LIN {X 0,Y 276.672,Z 702.695,A -85,B 0,C 180,E1 10836.654,E2 10836.654} C_VEL
LIN {X 0,Y 284.266,Z 684.369,A -85,B 0,C 180,E1 10834.788,E2 10834.788} C_VEL
LIN {X 0,Y 290.74,Z 666.187,A -85,B 0,C 180,E1 10833.316,E2 10833.316} C_VEL
LIN {X 0,Y 296.314,Z 647.189,A -85,B 0,C 180,E1 10832.121,E2 10832.121} C_VEL
LIN {X 0,Y 301.073,Z 626.782,A -85,B 0,C 180,E1 10831.146,E2 10831.146} C_VEL
LIN {X 0,Y 304.823,Z 604.834,A -85,B 0,C 180,E1 10830.396,E2 10830.396} C_VEL
LIN {X 0,Y 307.244,Z 581.509,A -85,B 0,C 180,E1 10829.851,E2 10829.851} C_VEL
LIN {X 0,Y 318.567,Z 436.926,A -85,B 0,C 180,E1 10826.925,E2 10826.925} C_VEL
LIN {X 0,Y 313.607,Z 427.1,A -85,B 0,C 180,E1 10824.286,E2 10824.286} C_VEL
LIN {X 0,Y 310.865,Z 421.791,A -85,B 0,C 180,E1 10822.654,E2 10822.654} C_VEL
LIN {X 0,Y 308.904,Z 419.239,A -85,B 0,C 180,E1 10821.467,E2 10821.467} C_VEL
LIN {X 0,Y 305.636,Z 417.774,A -85,B 0,C 180,E1 10819.49,E2 10819.49} C_VEL
LIN {X 0,Y 302.26,Z 416.33,A -85,B 0,C 180,E1 10817.137,E2 10817.137} C_VEL
LIN {X 0,Y 301.335,Z 415.075,A -85,B 0,C 180,E1 10816.335,E2 10816.335} C_VEL
LIN {X 0,Y 298.276,Z 409.863,A -85,B 0,C 180,E1 10813.078,E2 10813.078} C_VEL
LIN {X 0,Y 296.354,Z 406.465,A -85,B 0,C 180,E1 10810.301,E2 10810.301} C_VEL
LIN {X 0,Y 294.296,Z 402.303,A -85,B 0,C 180,E1 10804.677,E2 10804.677} C_VEL
LIN {X 0,Y 294.445,Z 402.242,A -85,B 0,C 180,E1 10799.611,E2 10799.611} C_VEL
LIN {X 0,Y 294.991,Z 403.216,A -85,B 0,C 180,E1 10797.669,E2 10797.669} C_VEL
LIN {X 0,Y 297.892,Z 407.607,A -85,B 0,C 180,E1 10792.479,E2 10792.479} C_VEL
LIN {X 0,Y 300.923,Z 412.517,A -85,B 0,C 180,E1 10789.083,E2 10789.083} C_VEL
LIN {X 0,Y 304.112,Z 417.715,A -85,B 0,C 180,E1 10786.307,E2 10786.307} C_VEL
LIN {X 0,Y 308.123,Z 424.469,A -85,B 0,C 180,E1 10783.408,E2 10783.408} C_VEL
LIN {X 0,Y 313.319,Z 434.005,A -85,B 0,C 180,E1 10780.229,E2 10780.229} C_VEL
LIN {X 0,Y 316.208,Z 439.917,A -85,B 0,C 180,E1 10778.643,E2 10778.643} C_VEL
LIN {X 0,Y 301.942,Z 602.181,A -85,B 0,C 180,E1 10775.206,E2 10775.206} C_VEL
LIN {X 0,Y 298.426,Z 624.101,A -85,B 0,C 180,E1 10774.558,E2 10774.558} C_VEL
LIN {X 0,Y 293.62,Z 645.542,A -85,B 0,C 180,E1 10773.691,E2 10773.691} C_VEL
LIN {X 0,Y 287.814,Z 666.096,A -85,B 0,C 180,E1 10772.57,E2 10772.57} C_VEL
LIN {X 0,Y 280.882,Z 686.418,A -85,B 0,C 180,E1 10771.123,E2 10771.123} C_VEL
LIN {X 0,Y 273.081,Z 705.676,A -85,B 0,C 180,E1 10769.362,E2 10769.362} C_VEL
LIN {X 0,Y 264.582,Z 724.162,A -85,B 0,C 180,E1 10767.225,E2 10767.225} C_VEL
LIN {X 0,Y 255.528,Z 741.796,A -85,B 0,C 180,E1 10764.668,E2 10764.668} C_VEL
LIN {X 0,Y 246.449,Z 757.992,A -85,B 0,C 180,E1 10761.722,E2 10761.722} C_VEL
LIN {X 0,Y 237.249,Z 773.128,A -85,B 0,C 180,E1 10758.239,E2 10758.239} C_VEL
LIN {X 0,Y 228.73,Z 786.502,A -85,B 0,C 180,E1 10754.378,E2 10754.378} C_VEL
LIN {X 0,Y 220.859,Z 798.628,A -85,B 0,C 180,E1 10750.003,E2 10750.003} C_VEL
LIN {X 0,Y 213.914,Z 809.4,A -85,B 0,C 180,E1 10745.093,E2 10745.093} C_VEL
LIN {X 0,Y 208.157,Z 818.76,A -85,B 0,C 180,E1 10739.61,E2 10739.61} C_VEL
LIN {X 0,Y 203.936,Z 826.542,A -85,B 0,C 180,E1 10733.704,E2 10733.704} C_VEL
LIN {X 0,Y 201.477,Z 832.324,A -85,B 0,C 180,E1 10727.919,E2 10727.919} C_VEL
LIN {X 0,Y 200.346,Z 836.379,A -85,B 0,C 180,E1 10722.099,E2 10722.099} C_VEL
LIN {X 0,Y 200.15,Z 838.918,A -85,B 0,C 180,E1 10716.309,E2 10716.309} C_VEL
LIN {X 0,Y 200.239,Z 839.79,A -85,B 0,C 180,E1 10711.717,E2 10711.717} C_VEL
LIN {X 0,Y 200.223,Z 839.71,A -85,B 0,C 180,E1 10707.424,E2 10707.424} C_VEL
LIN {X 0,Y 200.147,Z 838.438,A -85,B 0,C 180,E1 10702.248,E2 10702.248} C_VEL
LIN {X 0,Y 200.445,Z 835.835,A -85,B 0,C 180,E1 10697.029,E2 10697.029} C_VEL
LIN {X 0,Y 201.851,Z 831.232,A -85,B 0,C 180,E1 10690.918,E2 10690.918} C_VEL
LIN {X 0,Y 204.615,Z 825.211,A -85,B 0,C 180,E1 10685.151,E2 10685.151} C_VEL
LIN {X 0,Y 209.018,Z 817.23,A -85,B 0,C 180,E1 10679.433,E2 10679.433} C_VEL
LIN {X 0,Y 215.251,Z 807.171,A -85,B 0,C 180,E1 10673.849,E2 10673.849} C_VEL
LIN {X 0,Y 222.494,Z 796.02,A -85,B 0,C 180,E1 10668.998,E2 10668.998} C_VEL
LIN {X 0,Y 230.974,Z 782.987,A -85,B 0,C 180,E1 10664.529,E2 10664.529} C_VEL
LIN {X 0,Y 239.928,Z 768.64,A -85,B 0,C 180,E1 10660.674,E2 10660.674} C_VEL
LIN {X 0,Y 249.093,Z 753.165,A -85,B 0,C 180,E1 10657.369,E2 10657.369} C_VEL
LIN {X 0,Y 258.358,Z 736.244,A -85,B 0,C 180,E1 10654.483,E2 10654.483} C_VEL
LIN {X 0,Y 267.078,Z 718.805,A -85,B 0,C 180,E1 10652.113,E2 10652.113} C_VEL
LIN {X 0,Y 275.548,Z 699.551,A -85,B 0,C 180,E1 10650.049,E2 10650.049} C_VEL
LIN {X 0,Y 283.028,Z 679.99,A -85,B 0,C 180,E1 10648.403,E2 10648.403} C_VEL
LIN {X 0,Y 289.656,Z 659.53,A -85,B 0,C 180,E1 10647.056,E2 10647.056} C_VEL
LIN {X 0,Y 295.215,Z 638.606,A -85,B 0,C 180,E1 10646.008,E2 10646.008} C_VEL
LIN {X 0,Y 299.653,Z 616.702,A -85,B 0,C 180,E1 10645.216,E2 10645.216} C_VEL
LIN {X 0,Y 302.559,Z 594.85,A -85,B 0,C 180,E1 10644.635,E2 10644.635} C_VEL
LIN {X 0,Y 316.03,Z 439.44,A -85,B 0,C 180,E1 10641.336,E2 10641.336} C_VEL
LIN {X 0,Y 310.546,Z 428.999,A -85,B 0,C 180,E1 10638.247,E2 10638.247} C_VEL
LIN {X 0,Y 305.934,Z 420.872,A -85,B 0,C 180,E1 10635.205,E2 10635.205} C_VEL
LIN {X 0,Y 302.263,Z 414.828,A -85,B 0,C 180,E1 10632.319,E2 10632.319} C_VEL
LIN {X 0,Y 299.8,Z 410.85,A -85,B 0,C 180,E1 10629.987,E2 10629.987} C_VEL
LIN {X 0,Y 297.263,Z 406.753,A -85,B 0,C 180,E1 10626.955,E2 10626.955} C_VEL
LIN {X 0,Y 294.455,Z 402.282,A -85,B 0,C 180,E1 10621.362,E2 10621.362} C_VEL
LIN {X 0,Y 293.88,Z 401.961,A -85,B 0,C 180,E1 10616.489,E2 10616.489} C_VEL
LIN {X 0,Y 294.254,Z 402.624,A -85,B 0,C 180,E1 10614.149,E2 10614.149} C_VEL
LIN {X 0,Y 296.669,Z 407.215,A -85,B 0,C 180,E1 10608.727,E2 10608.727} C_VEL
LIN {X 0,Y 299.047,Z 411.383,A -85,B 0,C 180,E1 10605.675,E2 10605.675} C_VEL
LIN {X 0,Y 301.903,Z 416.413,A -85,B 0,C 180,E1 10602.857,E2 10602.857} C_VEL
LIN {X 0,Y 305.778,Z 423.433,A -85,B 0,C 180,E1 10599.774,E2 10599.774} C_VEL
LIN {X 0,Y 310.068,Z 431.486,A -85,B 0,C 180,E1 10596.933,E2 10596.933} C_VEL
LIN {X 0,Y 314.826,Z 441.211,A -85,B 0,C 180,E1 10594.2,E2 10594.2} C_VEL
LIN {X 0,Y 301.88,Z 598.214,A -85,B 0,C 180,E1 10591.019,E2 10591.019} C_VEL
LIN {X 0,Y 298.541,Z 619.734,A -85,B 0,C 180,E1 10590.375,E2 10590.375} C_VEL
LIN {X 0,Y 294.115,Z 639.956,A -85,B 0,C 180,E1 10589.515,E2 10589.515} C_VEL
LIN {X 0,Y 288.351,Z 660.439,A -85,B 0,C 180,E1 10588.348,E2 10588.348} C_VEL
LIN {X 0,Y 282.015,Z 678.968,A -85,B 0,C 180,E1 10586.978,E2 10586.978} C_VEL
LIN {X 0,Y 274.458,Z 697.523,A -85,B 0,C 180,E1 10585.231,E2 10585.231} C_VEL
LIN {X 0,Y 266.516,Z 714.386,A -85,B 0,C 180,E1 10583.22,E2 10583.22} C_VEL
LIN {X 0,Y 257.664,Z 731.079,A -85,B 0,C 180,E1 10580.727,E2 10580.727} C_VEL
LIN {X 0,Y 249.019,Z 745.804,A -85,B 0,C 180,E1 10577.97,E2 10577.97} C_VEL
LIN {X 0,Y 240.155,Z 759.6,A -85,B 0,C 180,E1 10574.716,E2 10574.716} C_VEL
LIN {X 0,Y 231.593,Z 771.968,A -85,B 0,C 180,E1 10571.012,E2 10571.012} C_VEL
LIN {X 0,Y 223.172,Z 783.563,A -85,B 0,C 180,E1 10566.573,E2 10566.573} C_VEL
LIN {X 0,Y 216.051,Z 793.13,A -85,B 0,C 180,E1 10561.841,E2 10561.841} C_VEL
LIN {X 0,Y 210.056,Z 801.285,A -85,B 0,C 180,E1 10556.578,E2 10556.578} C_VEL
LIN {X 0,Y 205.429,Z 807.855,A -85,B 0,C 180,E1 10550.811,E2 10550.811} C_VEL
LIN {X 0,Y 202.547,Z 812.407,A -85,B 0,C 180,E1 10545.166,E2 10545.166} C_VEL
LIN {X 0,Y 200.948,Z 815.59,A -85,B 0,C 180,E1 10539.162,E2 10539.162} C_VEL
LIN {X 0,Y 200.4,Z 817.13,A -85,B 0,C 180,E1 10533.719,E2 10533.719} C_VEL
LIN {X 0,Y 200.332,Z 817.331,A -85,B 0,C 180,E1 10528.284,E2 10528.284} C_VEL
LIN {X 0,Y 200.659,Z 816.383,A -85,B 0,C 180,E1 10522.844,E2 10522.844} C_VEL
LIN {X 0,Y 201.767,Z 813.901,A -85,B 0,C 180,E1 10517.115,E2 10517.115} C_VEL
LIN {X 0,Y 204.211,Z 809.715,A -85,B 0,C 180,E1 10511.147,E2 10511.147} C_VEL
LIN {X 0,Y 208.255,Z 803.795,A -85,B 0,C 180,E1 10505.311,E2 10505.311} C_VEL
LIN {X 0,Y 213.728,Z 796.374,A -85,B 0,C 180,E1 10499.937,E2 10499.937} C_VEL
LIN {X 0,Y 220.68,Z 787.067,A -85,B 0,C 180,E1 10494.873,E2 10494.873} C_VEL
LIN {X 0,Y 228.684,Z 776.16,A -85,B 0,C 180,E1 10490.333,E2 10490.333} C_VEL
LIN {X 0,Y 237.414,Z 763.748,A -85,B 0,C 180,E1 10486.318,E2 10486.318} C_VEL
LIN {X 0,Y 246.597,Z 749.809,A -85,B 0,C 180,E1 10482.789,E2 10482.789} C_VEL
LIN {X 0,Y 255.391,Z 735.349,A -85,B 0,C 180,E1 10479.886,E2 10479.886} C_VEL
LIN {X 0,Y 264.448,Z 718.812,A -85,B 0,C 180,E1 10477.263,E2 10477.263} C_VEL
LIN {X 0,Y 272.637,Z 701.841,A -85,B 0,C 180,E1 10475.135,E2 10475.135} C_VEL
LIN {X 0,Y 280.359,Z 683.561,A -85,B 0,C 180,E1 10473.314,E2 10473.314} C_VEL
LIN {X 0,Y 287.141,Z 664.723,A -85,B 0,C 180,E1 10471.831,E2 10471.831} C_VEL
LIN {X 0,Y 293.069,Z 644.824,A -85,B 0,C 180,E1 10470.619,E2 10470.619} C_VEL
LIN {X 0,Y 297.928,Z 623.713,A -85,B 0,C 180,E1 10469.666,E2 10469.666} C_VEL
LIN {X 0,Y 301.373,Z 603.001,A -85,B 0,C 180,E1 10469.003,E2 10469.003} C_VEL
LIN {X 0,Y 304.114,Z 575.028,A -85,B 0,C 180,E1 10468.38,E2 10468.38} C_VEL
LIN {X 0,Y 314.952,Z 441.247,A -85,B 0,C 180,E1 10465.68,E2 10465.68} C_VEL
LIN {X 0,Y 309.851,Z 430.902,A -85,B 0,C 180,E1 10462.732,E2 10462.732} C_VEL
LIN {X 0,Y 305.331,Z 422.359,A -85,B 0,C 180,E1 10459.663,E2 10459.663} C_VEL
LIN {X 0,Y 301.335,Z 415.075,A -85,B 0,C 180,E1 10456.335,E2 10456.335} C_VEL
LIN {X 0,Y 299.91,Z 413.527,A -85,B 0,C 180,E1 10455.028,E2 10455.028} C_VEL
LIN {X 0,Y 297.669,Z 413.637,A -85,B 0,C 180,E1 10452.932,E2 10452.932} C_VEL
LIN {X 0,Y 295.352,Z 414.27,A -85,B 0,C 180,E1 10450.238,E2 10450.238} C_VEL
LIN {X 0,Y 294.955,Z 413.941,A -85,B 0,C 180,E1 10449.588,E2 10449.588} C_VEL
LIN {X 0,Y 293.289,Z 410.213,A -85,B 0,C 180,E1 10444.498,E2 10444.498} C_VEL
LIN {X 0,Y 293.469,Z 410.189,A -85,B 0,C 180,E1 10439.61,E2 10439.61} C_VEL
LIN {X 0,Y 293.995,Z 411.255,A -85,B 0,C 180,E1 10437.661,E2 10437.661} C_VEL
LIN {X 0,Y 296.603,Z 415.287,A -85,B 0,C 180,E1 10432.835,E2 10432.835} C_VEL
LIN {X 0,Y 299.526,Z 420.223,A -85,B 0,C 180,E1 10429.421,E2 10429.421} C_VEL
LIN {X 0,Y 302.511,Z 425.254,A -85,B 0,C 180,E1 10426.72,E2 10426.72} C_VEL
LIN {X 0,Y 306.399,Z 432.083,A -85,B 0,C 180,E1 10423.799,E2 10423.799} C_VEL
LIN {X 0,Y 311.167,Z 441.169,A -85,B 0,C 180,E1 10420.771,E2 10420.771} C_VEL
LIN {X 0,Y 312.661,Z 444.381,A -85,B 0,C 180,E1 10419.895,E2 10419.895} C_VEL
LIN {X 0,Y 298.397,Z 602.136,A -85,B 0,C 180,E1 10416.579,E2 10416.579} C_VEL
LIN {X 0,Y 294.778,Z 624.153,A -85,B 0,C 180,E1 10415.937,E2 10415.937} C_VEL
LIN {X 0,Y 289.915,Z 645.311,A -85,B 0,C 180,E1 10415.095,E2 10415.095} C_VEL
LIN {X 0,Y 284.02,Z 665.699,A -85,B 0,C 180,E1 10414.003,E2 10414.003} C_VEL
LIN {X 0,Y 277.026,Z 685.694,A -85,B 0,C 180,E1 10412.605,E2 10412.605} C_VEL
LIN {X 0,Y 268.993,Z 705.031,A -85,B 0,C 180,E1 10410.866,E2 10410.866} C_VEL
LIN {X 0,Y 260.257,Z 723.497,A -85,B 0,C 180,E1 10408.759,E2 10408.759} C_VEL
LIN {X 0,Y 251.17,Z 740.681,A -85,B 0,C 180,E1 10406.301,E2 10406.301} C_VEL
LIN {X 0,Y 241.439,Z 757.416,A -85,B 0,C 180,E1 10403.275,E2 10403.275} C_VEL
LIN {X 0,Y 231.794,Z 772.617,A -85,B 0,C 180,E1 10399.772,E2 10399.772} C_VEL
LIN {X 0,Y 222.858,Z 786.007,A -85,B 0,C 180,E1 10395.875,E2 10395.875} C_VEL
LIN {X 0,Y 214.358,Z 798.4,A -85,B 0,C 180,E1 10391.326,E2 10391.326} C_VEL
LIN {X 0,Y 206.806,Z 809.455,A -85,B 0,C 180,E1 10386.145,E2 10386.145} C_VEL
LIN {X 0,Y 200.684,Z 818.756,A -85,B 0,C 180,E1 10380.467,E2 10380.467} C_VEL
LIN {X 0,Y 196.215,Z 826.398,A -85,B 0,C 180,E1 10374.377,E2 10374.377} C_VEL
LIN {X 0,Y 193.482,Z 832.327,A -85,B 0,C 180,E1 10368.039,E2 10368.039} C_VEL
LIN {X 0,Y 192.362,Z 836.119,A -85,B 0,C 180,E1 10362.265,E2 10362.265} C_VEL
LIN {X 0,Y 192.16,Z 838.516,A -85,B 0,C 180,E1 10356.377,E2 10356.377} C_VEL
LIN {X 0,Y 192.25,Z 839.342,A -85,B 0,C 180,E1 10351.788,E2 10351.788} C_VEL
LIN {X 0,Y 192.232,Z 839.261,A -85,B 0,C 180,E1 10347.317,E2 10347.317} C_VEL
LIN {X 0,Y 192.155,Z 837.984,A -85,B 0,C 180,E1 10341.924,E2 10341.924} C_VEL
LIN {X 0,Y 192.511,Z 835.376,A -85,B 0,C 180,E1 10336.484,E2 10336.484} C_VEL
LIN {X 0,Y 194.094,Z 830.766,A -85,B 0,C 180,E1 10330.124,E2 10330.124} C_VEL
LIN {X 0,Y 197.134,Z 824.742,A -85,B 0,C 180,E1 10324.14,E2 10324.14} C_VEL
LIN {X 0,Y 201.816,Z 816.888,A -85,B 0,C 180,E1 10318.322,E2 10318.322} C_VEL
LIN {X 0,Y 208.214,Z 807.226,A -85,B 0,C 180,E1 10312.768,E2 10312.768} C_VEL
LIN {X 0,Y 215.835,Z 796.186,A -85,B 0,C 180,E1 10307.802,E2 10307.802} C_VEL
LIN {X 0,Y 224.689,Z 783.24,A -85,B 0,C 180,E1 10303.258,E2 10303.258} C_VEL
LIN {X 0,Y 234.032,Z 768.997,A -85,B 0,C 180,E1 10299.352,E2 10299.352} C_VEL
LIN {X 0,Y 243.538,Z 753.667,A -85,B 0,C 180,E1 10296.024,E2 10296.024} C_VEL
LIN {X 0,Y 252.791,Z 737.538,A -85,B 0,C 180,E1 10293.226,E2 10293.226} C_VEL
LIN {X 0,Y 261.927,Z 719.945,A -85,B 0,C 180,E1 10290.81,E2 10290.81} C_VEL
LIN {X 0,Y 270.412,Z 701.461,A -85,B 0,C 180,E1 10288.802,E2 10288.802} C_VEL
LIN {X 0,Y 278.49,Z 681.282,A -85,B 0,C 180,E1 10287.081,E2 10287.081} C_VEL
LIN {X 0,Y 285.281,Z 661.235,A -85,B 0,C 180,E1 10285.748,E2 10285.748} C_VEL
LIN {X 0,Y 291.071,Z 640.344,A -85,B 0,C 180,E1 10284.693,E2 10284.693} C_VEL
LIN {X 0,Y 295.632,Z 618.832,A -85,B 0,C 180,E1 10283.908,E2 10283.908} C_VEL
LIN {X 0,Y 298.847,Z 596.481,A -85,B 0,C 180,E1 10283.303,E2 10283.303} C_VEL
LIN {X 0,Y 312.496,Z 443.973,A -85,B 0,C 180,E1 10280.093,E2 10280.093} C_VEL
LIN {X 0,Y 307.033,Z 433.38,A -85,B 0,C 180,E1 10276.75,E2 10276.75} C_VEL
LIN {X 0,Y 302.666,Z 425.671,A -85,B 0,C 180,E1 10273.565,E2 10273.565} C_VEL
LIN {X 0,Y 300.202,Z 421.559,A -85,B 0,C 180,E1 10271.43,E2 10271.43} C_VEL
LIN {X 0,Y 298.341,Z 418.411,A -85,B 0,C 180,E1 10269.549,E2 10269.549} C_VEL
LIN {X 0,Y 295.99,Z 414.475,A -85,B 0,C 180,E1 10266.595,E2 10266.595} C_VEL
LIN {X 0,Y 293.418,Z 410.184,A -85,B 0,C 180,E1 10261.171,E2 10261.171} C_VEL
LIN {X 0,Y 292.92,Z 409.93,A -85,B 0,C 180,E1 10256.281,E2 10256.281} C_VEL
LIN {X 0,Y 293.277,Z 410.644,A -85,B 0,C 180,E1 10254.129,E2 10254.129} C_VEL
LIN {X 0,Y 295.499,Z 415.05,A -85,B 0,C 180,E1 10248.978,E2 10248.978} C_VEL
LIN {X 0,Y 297.683,Z 419.005,A -85,B 0,C 180,E1 10246.067,E2 10246.067} C_VEL
LIN {X 0,Y 300.402,Z 423.986,A -85,B 0,C 180,E1 10243.267,E2 10243.267} C_VEL
LIN {X 0,Y 304.105,Z 430.961,A -85,B 0,C 180,E1 10240.205,E2 10240.205} C_VEL
LIN {X 0,Y 308.117,Z 438.851,A -85,B 0,C 180,E1 10237.435,E2 10237.435} C_VEL
LIN {X 0,Y 311.346,Z 445.782,A -85,B 0,C 180,E1 10235.461,E2 10235.461} C_VEL
LIN {X 0,Y 298.336,Z 598.392,A -85,B 0,C 180,E1 10232.39,E2 10232.39} C_VEL
LIN {X 0,Y 294.913,Z 619.881,A -85,B 0,C 180,E1 10231.754,E2 10231.754} C_VEL
LIN {X 0,Y 290.352,Z 640.196,A -85,B 0,C 180,E1 10230.902,E2 10230.902} C_VEL
LIN {X 0,Y 284.254,Z 661.228,A -85,B 0,C 180,E1 10229.714,E2 10229.714} C_VEL
LIN {X 0,Y 277.387,Z 680.531,A -85,B 0,C 180,E1 10228.283,E2 10228.283} C_VEL
LIN {X 0,Y 269.638,Z 698.933,A -85,B 0,C 180,E1 10226.544,E2 10226.544} C_VEL
LIN {X 0,Y 261.13,Z 716.273,A -85,B 0,C 180,E1 10224.452,E2 10224.452} C_VEL
LIN {X 0,Y 252.017,Z 732.702,A -85,B 0,C 180,E1 10221.953,E2 10221.953} C_VEL
LIN {X 0,Y 242.501,Z 748.118,A -85,B 0,C 180,E1 10218.982,E2 10218.982} C_VEL
LIN {X 0,Y 233.387,Z 761.659,A -85,B 0,C 180,E1 10215.678,E2 10215.678} C_VEL
LIN {X 0,Y 224.074,Z 774.491,A -85,B 0,C 180,E1 10211.67,E2 10211.67} C_VEL
LIN {X 0,Y 215.443,Z 785.693,A -85,B 0,C 180,E1 10207.107,E2 10207.107} C_VEL
LIN {X 0,Y 208.146,Z 794.915,A -85,B 0,C 180,E1 10202.221,E2 10202.221} C_VEL
LIN {X 0,Y 201.748,Z 803.09,A -85,B 0,C 180,E1 10196.489,E2 10196.489} C_VEL
LIN {X 0,Y 197.317,Z 809.099,A -85,B 0,C 180,E1 10190.775,E2 10190.775} C_VEL
LIN {X 0,Y 194.333,Z 813.638,A -85,B 0,C 180,E1 10184.602,E2 10184.602} C_VEL
LIN {X 0,Y 192.875,Z 816.357,A -85,B 0,C 180,E1 10178.646,E2 10178.646} C_VEL
LIN {X 0,Y 192.376,Z 817.707,A -85,B 0,C 180,E1 10172.681,E2 10172.681} C_VEL
LIN {X 0,Y 192.36,Z 817.738,A -85,B 0,C 180,E1 10167.617,E2 10167.617} C_VEL
LIN {X 0,Y 192.82,Z 816.515,A -85,B 0,C 180,E1 10161.652,E2 10161.652} C_VEL
LIN {X 0,Y 194.206,Z 813.905,A -85,B 0,C 180,E1 10155.693,E2 10155.693} C_VEL
LIN {X 0,Y 197.084,Z 809.449,A -85,B 0,C 180,E1 10149.51,E2 10149.51} C_VEL
LIN {X 0,Y 201.68,Z 803.242,A -85,B 0,C 180,E1 10143.501,E2 10143.501} C_VEL
LIN {X 0,Y 208.081,Z 795.087,A -85,B 0,C 180,E1 10137.749,E2 10137.749} C_VEL
LIN {X 0,Y 215.341,Z 785.936,A -85,B 0,C 180,E1 10132.872,E2 10132.872} C_VEL
LIN {X 0,Y 223.961,Z 774.775,A -85,B 0,C 180,E1 10128.304,E2 10128.304} C_VEL
LIN {X 0,Y 233.265,Z 761.979,A -85,B 0,C 180,E1 10124.291,E2 10124.291} C_VEL
LIN {X 0,Y 242.368,Z 748.5,A -85,B 0,C 180,E1 10120.982,E2 10120.982} C_VEL
LIN {X 0,Y 252.198,Z 732.614,A -85,B 0,C 180,E1 10117.915,E2 10117.915} C_VEL
LIN {X 0,Y 260.995,Z 716.818,A -85,B 0,C 180,E1 10115.506,E2 10115.506} C_VEL
LIN {X 0,Y 269.497,Z 699.536,A -85,B 0,C 180,E1 10113.411,E2 10113.411} C_VEL
LIN {X 0,Y 277.246,Z 681.252,A -85,B 0,C 180,E1 10111.67,E2 10111.67} C_VEL
LIN {X 0,Y 284.112,Z 662.135,A -85,B 0,C 180,E1 10110.237,E2 10110.237} C_VEL
LIN {X 0,Y 290.004,Z 642.19,A -85,B 0,C 180,E1 10109.087,E2 10109.087} C_VEL
LIN {X 0,Y 294.803,Z 621.393,A -85,B 0,C 180,E1 10108.192,E2 10108.192} C_VEL
LIN {X 0,Y 298.306,Z 599.8,A -85,B 0,C 180,E1 10107.541,E2 10107.541} C_VEL
LIN {X 0,Y 302.156,Z 556.981,A -85,B 0,C 180,E1 10106.647,E2 10106.647} C_VEL
LIN {X 0,Y 311.488,Z 445.629,A -85,B 0,C 180,E1 10104.411,E2 10104.411} C_VEL
LIN {X 0,Y 306.307,Z 434.97,A -85,B 0,C 180,E1 10101.143,E2 10101.143} C_VEL
LIN {X 0,Y 302.014,Z 426.745,A -85,B 0,C 180,E1 10097.883,E2 10097.883} C_VEL
LIN {X 0,Y 299.225,Z 421.673,A -85,B 0,C 180,E1 10095.307,E2 10095.307} C_VEL
LIN {X 0,Y 296.924,Z 417.455,A -85,B 0,C 180,E1 10092.644,E2 10092.644} C_VEL
LIN {X 0,Y 295.16,Z 414.211,A -85,B 0,C 180,E1 10089.949,E2 10089.949} C_VEL
LIN {X 0,Y 294.955,Z 413.941,A -85,B 0,C 180,E1 10089.588,E2 10089.588} C_VEL
LIN {X 0,Y 294.052,Z 413.81,A -85,B 0,C 180,E1 10087.976,E2 10087.976} C_VEL
LIN {X 0,Y 292.202,Z 417.825,A -85,B 0,C 180,E1 10083.327,E2 10083.327} C_VEL
LIN {X 0,Y 292.155,Z 417.945,A -85,B 0,C 180,E1 10082.665,E2 10082.665} C_VEL
LIN {X 0,Y 292.731,Z 418.491,A -85,B 0,C 180,E1 10078.63,E2 10078.63} C_VEL
LIN {X 0,Y 295.393,Z 423.114,A -85,B 0,C 180,E1 10073.099,E2 10073.099} C_VEL
LIN {X 0,Y 298.141,Z 427.926,A -85,B 0,C 180,E1 10069.762,E2 10069.762} C_VEL
LIN {X 0,Y 301.142,Z 433.176,A -85,B 0,C 180,E1 10066.952,E2 10066.952} C_VEL
LIN {X 0,Y 305.407,Z 441.02,A -85,B 0,C 180,E1 10063.696,E2 10063.696} C_VEL
LIN {X 0,Y 309.261,Z 448.958,A -85,B 0,C 180,E1 10061.174,E2 10061.174} C_VEL
LIN {X 0,Y 295.041,Z 601.989,A -85,B 0,C 180,E1 10057.987,E2 10057.987} C_VEL
LIN {X 0,Y 291.349,Z 623.97,A -85,B 0,C 180,E1 10057.357,E2 10057.357} C_VEL
LIN {X 0,Y 286.539,Z 644.522,A -85,B 0,C 180,E1 10056.56,E2 10056.56} C_VEL
LIN {X 0,Y 280.683,Z 664.509,A -85,B 0,C 180,E1 10055.523,E2 10055.523} C_VEL
LIN {X 0,Y 273.361,Z 684.962,A -85,B 0,C 180,E1 10054.126,E2 10054.126} C_VEL
LIN {X 0,Y 265.466,Z 703.562,A -85,B 0,C 180,E1 10052.495,E2 10052.495} C_VEL
LIN {X 0,Y 256.046,Z 722.99,A -85,B 0,C 180,E1 10050.324,E2 10050.324} C_VEL
LIN {X 0,Y 246.684,Z 740.136,A -85,B 0,C 180,E1 10047.897,E2 10047.897} C_VEL
LIN {X 0,Y 236.816,Z 756.502,A -85,B 0,C 180,E1 10044.957,E2 10044.957} C_VEL
LIN {X 0,Y 227.099,Z 771.235,A -85,B 0,C 180,E1 10041.597,E2 10041.597} C_VEL
LIN {X 0,Y 217.143,Z 785.515,A -85,B 0,C 180,E1 10037.452,E2 10037.452} C_VEL
LIN {X 0,Y 208.368,Z 797.663,A -85,B 0,C 180,E1 10032.951,E2 10032.951} C_VEL
LIN {X 0,Y 200.139,Z 808.976,A -85,B 0,C 180,E1 10027.551,E2 10027.551} C_VEL
LIN {X 0,Y 193.629,Z 818.185,A -85,B 0,C 180,E1 10021.782,E2 10021.782} C_VEL
LIN {X 0,Y 188.712,Z 825.932,A -85,B 0,C 180,E1 10015.414,E2 10015.414} C_VEL
LIN {X 0,Y 185.697,Z 831.849,A -85,B 0,C 180,E1 10008.848,E2 10008.848} C_VEL
LIN {X 0,Y 184.423,Z 835.639,A -85,B 0,C 180,E1 10002.843,E2 10002.843} C_VEL
LIN {X 0,Y 184.172,Z 838.016,A -85,B 0,C 180,E1 9996.859,E2 9996.859} C_VEL
LIN {X 0,Y 184.26,Z 838.893,A -85,B 0,C 180,E1 9991.866,E2 9991.866} C_VEL
LIN {X 0,Y 184.241,Z 838.812,A -85,B 0,C 180,E1 9987.201,E2 9987.201} C_VEL
LIN {X 0,Y 184.164,Z 837.53,A -85,B 0,C 180,E1 9981.571,E2 9981.571} C_VEL
LIN {X 0,Y 184.6,Z 834.875,A -85,B 0,C 180,E1 9975.816,E2 9975.816} C_VEL
LIN {X 0,Y 186.377,Z 830.302,A -85,B 0,C 180,E1 9969.264,E2 9969.264} C_VEL
LIN {X 0,Y 189.922,Z 823.931,A -85,B 0,C 180,E1 9962.742,E2 9962.742} C_VEL
LIN {X 0,Y 195.389,Z 815.559,A -85,B 0,C 180,E1 9956.451,E2 9956.451} C_VEL
LIN {X 0,Y 202.418,Z 805.667,A -85,B 0,C 180,E1 9950.784,E2 9950.784} C_VEL
LIN {X 0,Y 211.142,Z 793.712,A -85,B 0,C 180,E1 9945.506,E2 9945.506} C_VEL
LIN {X 0,Y 220.329,Z 780.934,A -85,B 0,C 180,E1 9941.124,E2 9941.124} C_VEL
LIN {X 0,Y 230.061,Z 766.742,A -85,B 0,C 180,E1 9937.316,E2 9937.316} C_VEL
LIN {X 0,Y 239.727,Z 751.568,A -85,B 0,C 180,E1 9934.118,E2 9934.118} C_VEL
LIN {X 0,Y 249.731,Z 734.476,A -85,B 0,C 180,E1 9931.265,E2 9931.265} C_VEL
LIN {X 0,Y 258.926,Z 717.112,A -85,B 0,C 180,E1 9928.976,E2 9928.976} C_VEL
LIN {X 0,Y 267.687,Z 698.335,A -85,B 0,C 180,E1 9927.024,E2 9927.024} C_VEL
LIN {X 0,Y 275.285,Z 679.439,A -85,B 0,C 180,E1 9925.486,E2 9925.486} C_VEL
LIN {X 0,Y 282.234,Z 659.05,A -85,B 0,C 180,E1 9924.187,E2 9924.187} C_VEL
LIN {X 0,Y 288.035,Z 638.224,A -85,B 0,C 180,E1 9923.183,E2 9923.183} C_VEL
LIN {X 0,Y 292.661,Z 616.369,A -85,B 0,C 180,E1 9922.421,E2 9922.421} C_VEL
LIN {X 0,Y 295.703,Z 594.476,A -85,B 0,C 180,E1 9921.854,E2 9921.854} C_VEL
LIN {X 0,Y 309.094,Z 448.662,A -85,B 0,C 180,E1 9918.824,E2 9918.824} C_VEL
LIN {X 0,Y 304.463,Z 439.409,A -85,B 0,C 180,E1 9915.768,E2 9915.768} C_VEL
LIN {X 0,Y 300.631,Z 432.429,A -85,B 0,C 180,E1 9912.777,E2 9912.777} C_VEL
LIN {X 0,Y 297.251,Z 426.439,A -85,B 0,C 180,E1 9909.486,E2 9909.486} C_VEL
LIN {X 0,Y 294.73,Z 422.195,A -85,B 0,C 180,E1 9906.232,E2 9906.232} C_VEL
LIN {X 0,Y 292.385,Z 418.086,A -85,B 0,C 180,E1 9900.979,E2 9900.979} C_VEL
LIN {X 0,Y 291.947,Z 417.874,A -85,B 0,C 180,E1 9896.269,E2 9896.269} C_VEL
LIN {X 0,Y 292.256,Z 418.529,A -85,B 0,C 180,E1 9894.306,E2 9894.306} C_VEL
LIN {X 0,Y 294.284,Z 422.75,A -85,B 0,C 180,E1 9889.329,E2 9889.329} C_VEL
LIN {X 0,Y 296.348,Z 426.669,A -85,B 0,C 180,E1 9886.438,E2 9886.438} C_VEL
LIN {X 0,Y 298.916,Z 431.556,A -85,B 0,C 180,E1 9883.681,E2 9883.681} C_VEL
LIN {X 0,Y 302.378,Z 438.355,A -85,B 0,C 180,E1 9880.69,E2 9880.69} C_VEL
LIN {X 0,Y 306.124,Z 446.059,A -85,B 0,C 180,E1 9877.988,E2 9877.988} C_VEL
LIN {X 0,Y 308.018,Z 450.255,A -85,B 0,C 180,E1 9876.755,E2 9876.755} C_VEL
LIN {X 0,Y 294.99,Z 598.371,A -85,B 0,C 180,E1 9873.796,E2 9873.796} C_VEL
LIN {X 0,Y 291.512,Z 619.754,A -85,B 0,C 180,E1 9873.175,E2 9873.175} C_VEL
LIN {X 0,Y 286.956,Z 639.699,A -85,B 0,C 180,E1 9872.359,E2 9872.359} C_VEL
LIN {X 0,Y 281.08,Z 659.775,A -85,B 0,C 180,E1 9871.262,E2 9871.262} C_VEL
LIN {X 0,Y 274.221,Z 678.933,A -85,B 0,C 180,E1 9869.898,E2 9869.898} C_VEL
LIN {X 0,Y 266.379,Z 697.18,A -85,B 0,C 180,E1 9868.228,E2 9868.228} C_VEL
LIN {X 0,Y 257.925,Z 714.221,A -85,B 0,C 180,E1 9866.253,E2 9866.253} C_VEL
LIN {X 0,Y 248.458,Z 731.057,A -85,B 0,C 180,E1 9863.788,E2 9863.788} C_VEL
LIN {X 0,Y 239.157,Z 745.908,A -85,B 0,C 180,E1 9861.041,E2 9861.041} C_VEL
LIN {X 0,Y 228.961,Z 760.595,A -85,B 0,C 180,E1 9857.561,E2 9857.561} C_VEL
LIN {X 0,Y 219.639,Z 772.931,A -85,B 0,C 180,E1 9853.783,E2 9853.783} C_VEL
LIN {X 0,Y 210.452,Z 784.409,A -85,B 0,C 180,E1 9849.247,E2 9849.247} C_VEL
LIN {X 0,Y 202.449,Z 794.056,A -85,B 0,C 180,E1 9844.264,E2 9844.264} C_VEL
LIN {X 0,Y 195.685,Z 802.201,A -85,B 0,C 180,E1 9838.704,E2 9838.704} C_VEL
LIN {X 0,Y 190.376,Z 808.771,A -85,B 0,C 180,E1 9832.544,E2 9832.544} C_VEL
LIN {X 0,Y 186.885,Z 813.511,A -85,B 0,C 180,E1 9826.153,E2 9826.153} C_VEL
LIN {X 0,Y 185.048,Z 816.597,A -85,B 0,C 180,E1 9819.642,E2 9819.642} C_VEL
LIN {X 0,Y 184.426,Z 818.088,A -85,B 0,C 180,E1 9813.73,E2 9813.73} C_VEL
LIN {X 0,Y 184.36,Z 818.227,A -85,B 0,C 180,E1 9808.135,E2 9808.135} C_VEL
LIN {X 0,Y 184.757,Z 817.283,A -85,B 0,C 180,E1 9802.225,E2 9802.225} C_VEL
LIN {X 0,Y 186.089,Z 814.803,A -85,B 0,C 180,E1 9796.008,E2 9796.008} C_VEL
LIN {X 0,Y 188.967,Z 810.623,A -85,B 0,C 180,E1 9789.561,E2 9789.561} C_VEL
LIN {X 0,Y 193.665,Z 804.674,A -85,B 0,C 180,E1 9783.275,E2 9783.275} C_VEL
LIN {X 0,Y 199.818,Z 797.337,A -85,B 0,C 180,E1 9777.629,E2 9777.629} C_VEL
LIN {X 0,Y 207.625,Z 787.991,A -85,B 0,C 180,E1 9772.296,E2 9772.296} C_VEL
LIN {X 0,Y 216.147,Z 777.485,A -85,B 0,C 180,E1 9767.743,E2 9767.743} C_VEL
LIN {X 0,Y 225.443,Z 765.461,A -85,B 0,C 180,E1 9763.706,E2 9763.706} C_VEL
LIN {X 0,Y 234.731,Z 752.618,A -85,B 0,C 180,E1 9760.32,E2 9760.32} C_VEL
LIN {X 0,Y 244.738,Z 737.439,A -85,B 0,C 180,E1 9757.19,E2 9757.19} C_VEL
LIN {X 0,Y 254.023,Z 721.691,A -85,B 0,C 180,E1 9754.652,E2 9754.652} C_VEL
LIN {X 0,Y 263.04,Z 704.47,A -85,B 0,C 180,E1 9752.453,E2 9752.453} C_VEL
LIN {X 0,Y 271.313,Z 686.358,A -85,B 0,C 180,E1 9750.629,E2 9750.629} C_VEL
LIN {X 0,Y 278.699,Z 667.385,A -85,B 0,C 180,E1 9749.126,E2 9749.126} C_VEL
LIN {X 0,Y 285.105,Z 647.198,A -85,B 0,C 180,E1 9747.904,E2 9747.904} C_VEL
LIN {X 0,Y 290.193,Z 626.832,A -85,B 0,C 180,E1 9746.979,E2 9746.979} C_VEL
LIN {X 0,Y 294.187,Z 605.052,A -85,B 0,C 180,E1 9746.272,E2 9746.272} C_VEL
LIN {X 0,Y 296.85,Z 581.323,A -85,B 0,C 180,E1 9745.734,E2 9745.734} C_VEL
LIN {X 0,Y 308.162,Z 450.154,A -85,B 0,C 180,E1 9743.116,E2 9743.116} C_VEL
LIN {X 0,Y 303.521,Z 440.303,A -85,B 0,C 180,E1 9739.935,E2 9739.935} C_VEL
LIN {X 0,Y 299.695,Z 432.82,A -85,B 0,C 180,E1 9736.769,E2 9736.769} C_VEL
LIN {X 0,Y 297.446,Z 428.647,A -85,B 0,C 180,E1 9734.516,E2 9734.516} C_VEL
LIN {X 0,Y 295.662,Z 425.157,A -85,B 0,C 180,E1 9732.302,E2 9732.302} C_VEL
LIN {X 0,Y 293.977,Z 421.954,A -85,B 0,C 180,E1 9729.594,E2 9729.594} C_VEL
LIN {X 0,Y 292.285,Z 418.126,A -85,B 0,C 180,E1 9724.316,E2 9724.316} C_VEL
LIN {X 0,Y 292.155,Z 417.945,A -85,B 0,C 180,E1 9722.665,E2 9722.665} C_VEL
LIN {X 0,Y 292.101,Z 418.899,A -85,B 0,C 180,E1 9721.264,E2 9721.264} C_VEL
LIN {X 0,Y 292.02,Z 422.577,A -85,B 0,C 180,E1 9719.304,E2 9719.304} C_VEL
LIN {X 0,Y 292.337,Z 427.67,A -85,B 0,C 180,E1 9716.829,E2 9716.829} C_VEL
LIN {X 0,Y 292.669,Z 428.684,A -85,B 0,C 180,E1 9715.97,E2 9715.97} C_VEL
LIN {X 0,Y 294.192,Z 430.94,A -85,B 0,C 180,E1 9713.365,E2 9713.365} C_VEL
LIN {X 0,Y 296.766,Z 435.627,A -85,B 0,C 180,E1 9710.106,E2 9710.106} C_VEL
LIN {X 0,Y 299.566,Z 440.711,A -85,B 0,C 180,E1 9707.372,E2 9707.372} C_VEL
LIN {X 0,Y 303.507,Z 448.281,A -85,B 0,C 180,E1 9704.23,E2 9704.23} C_VEL
LIN {X 0,Y 305.998,Z 453.748,A -85,B 0,C 180,E1 9702.476,E2 9702.476} C_VEL
LIN {X 0,Y 291.854,Z 601.952,A -85,B 0,C 180,E1 9699.424,E2 9699.424} C_VEL
LIN {X 0,Y 288.069,Z 623.974,A -85,B 0,C 180,E1 9698.803,E2 9698.803} C_VEL
LIN {X 0,Y 283.078,Z 644.754,A -85,B 0,C 180,E1 9698.013,E2 9698.013} C_VEL
LIN {X 0,Y 277.008,Z 664.861,A -85,B 0,C 180,E1 9696.984,E2 9696.984} C_VEL
LIN {X 0,Y 269.508,Z 685.249,A -85,B 0,C 180,E1 9695.611,E2 9695.611} C_VEL
LIN {X 0,Y 261.024,Z 704.569,A -85,B 0,C 180,E1 9693.926,E2 9693.926} C_VEL
LIN {X 0,Y 251.709,Z 723.087,A -85,B 0,C 180,E1 9691.863,E2 9691.863} C_VEL
LIN {X 0,Y 241.7,Z 740.73,A -85,B 0,C 180,E1 9689.364,E2 9689.364} C_VEL
LIN {X 0,Y 231.56,Z 756.917,A -85,B 0,C 180,E1 9686.443,E2 9686.443} C_VEL
LIN {X 0,Y 221.431,Z 771.598,A -85,B 0,C 180,E1 9683.055,E2 9683.055} C_VEL
LIN {X 0,Y 211.602,Z 785.021,A -85,B 0,C 180,E1 9679.114,E2 9679.114} C_VEL
LIN {X 0,Y 202.35,Z 797.182,A -85,B 0,C 180,E1 9674.558,E2 9674.558} C_VEL
LIN {X 0,Y 193.601,Z 808.497,A -85,B 0,C 180,E1 9669.054,E2 9669.054} C_VEL
LIN {X 0,Y 186.611,Z 817.712,A -85,B 0,C 180,E1 9663.127,E2 9663.127} C_VEL
LIN {X 0,Y 181.272,Z 825.466,A -85,B 0,C 180,E1 9656.536,E2 9656.536} C_VEL
LIN {X 0,Y 177.937,Z 831.388,A -85,B 0,C 180,E1 9649.703,E2 9649.703} C_VEL
LIN {X 0,Y 176.49,Z 835.182,A -85,B 0,C 180,E1 9643.431,E2 9643.431} C_VEL
LIN {X 0,Y 176.181,Z 837.641,A -85,B 0,C 180,E1 9636.845,E2 9636.845} C_VEL
LIN {X 0,Y 176.27,Z 838.445,A -85,B 0,C 180,E1 9631.95,E2 9631.95} C_VEL
LIN {X 0,Y 176.256,Z 838.39,A -85,B 0,C 180,E1 9627.399,E2 9627.399} C_VEL
LIN {X 0,Y 176.168,Z 837.316,A -85,B 0,C 180,E1 9621.843,E2 9621.843} C_VEL
LIN {X 0,Y 176.654,Z 834.555,A -85,B 0,C 180,E1 9615.431,E2 9615.431} C_VEL
LIN {X 0,Y 178.558,Z 830.109,A -85,B 0,C 180,E1 9608.656,E2 9608.656} C_VEL
LIN {X 0,Y 182.357,Z 823.806,A -85,B 0,C 180,E1 9601.867,E2 9601.867} C_VEL
LIN {X 0,Y 187.995,Z 815.753,A -85,B 0,C 180,E1 9595.524,E2 9595.524} C_VEL
LIN {X 0,Y 195.371,Z 806.037,A -85,B 0,C 180,E1 9589.688,E2 9589.688} C_VEL
LIN {X 0,Y 203.795,Z 795.2,A -85,B 0,C 180,E1 9584.653,E2 9584.653} C_VEL
LIN {X 0,Y 213.255,Z 782.729,A -85,B 0,C 180,E1 9580.163,E2 9580.163} C_VEL
LIN {X 0,Y 223.26,Z 768.843,A -85,B 0,C 180,E1 9576.283,E2 9576.283} C_VEL
LIN {X 0,Y 233.552,Z 753.58,A -85,B 0,C 180,E1 9572.935,E2 9572.935} C_VEL
LIN {X 0,Y 243.287,Z 737.907,A -85,B 0,C 180,E1 9570.209,E2 9570.209} C_VEL
LIN {X 0,Y 253.276,Z 719.911,A -85,B 0,C 180,E1 9567.763,E2 9567.763} C_VEL
LIN {X 0,Y 262.149,Z 701.805,A -85,B 0,C 180,E1 9565.829,E2 9565.829} C_VEL
LIN {X 0,Y 270.663,Z 681.831,A -85,B 0,C 180,E1 9564.158,E2 9564.158} C_VEL
LIN {X 0,Y 277.797,Z 662.055,A -85,B 0,C 180,E1 9562.871,E2 9562.871} C_VEL
LIN {X 0,Y 283.853,Z 641.338,A -85,B 0,C 180,E1 9561.853,E2 9561.853} C_VEL
LIN {X 0,Y 288.685,Z 620.008,A -85,B 0,C 180,E1 9561.09,E2 9561.09} C_VEL
LIN {X 0,Y 292.259,Z 596.843,A -85,B 0,C 180,E1 9560.474,E2 9560.474} C_VEL
LIN {X 0,Y 305.812,Z 453.301,A -85,B 0,C 180,E1 9557.505,E2 9557.505} C_VEL
LIN {X 0,Y 301.624,Z 444.773,A -85,B 0,C 180,E1 9554.493,E2 9554.493} C_VEL
LIN {X 0,Y 297.965,Z 437.876,A -85,B 0,C 180,E1 9551.321,E2 9551.321} C_VEL
LIN {X 0,Y 295.481,Z 433.527,A -85,B 0,C 180,E1 9548.66,E2 9548.66} C_VEL
LIN {X 0,Y 293.481,Z 429.913,A -85,B 0,C 180,E1 9545.866,E2 9545.866} C_VEL
LIN {X 0,Y 291.355,Z 425.99,A -85,B 0,C 180,E1 9540.786,E2 9540.786} C_VEL
LIN {X 0,Y 290.994,Z 425.843,A -85,B 0,C 180,E1 9536.059,E2 9536.059} C_VEL
LIN {X 0,Y 291.275,Z 426.557,A -85,B 0,C 180,E1 9534.286,E2 9534.286} C_VEL
LIN {X 0,Y 293.19,Z 430.715,A -85,B 0,C 180,E1 9529.487,E2 9529.487} C_VEL
LIN {X 0,Y 295.053,Z 434.396,A -85,B 0,C 180,E1 9526.777,E2 9526.777} C_VEL
LIN {X 0,Y 297.539,Z 439.316,A -85,B 0,C 180,E1 9524.004,E2 9524.004} C_VEL
LIN {X 0,Y 300.787,Z 445.98,A -85,B 0,C 180,E1 9521.088,E2 9521.088} C_VEL
LIN {X 0,Y 304.29,Z 453.563,A -85,B 0,C 180,E1 9518.457,E2 9518.457} C_VEL
LIN {X 0,Y 304.822,Z 455.055,A -85,B 0,C 180,E1 9518.07,E2 9518.07} C_VEL
LIN {X 0,Y 291.801,Z 598.543,A -85,B 0,C 180,E1 9515.23,E2 9515.23} C_VEL
LIN {X 0,Y 288.24,Z 619.913,A -85,B 0,C 180,E1 9514.62,E2 9514.62} C_VEL
LIN {X 0,Y 283.554,Z 639.938,A -85,B 0,C 180,E1 9513.816,E2 9513.816} C_VEL
LIN {X 0,Y 277.728,Z 659.44,A -85,B 0,C 180,E1 9512.774,E2 9512.774} C_VEL
LIN {X 0,Y 270.856,Z 678.277,A -85,B 0,C 180,E1 9511.467,E2 9511.467} C_VEL
LIN {X 0,Y 262.625,Z 697.013,A -85,B 0,C 180,E1 9509.792,E2 9509.792} C_VEL
LIN {X 0,Y 253.917,Z 714.138,A -85,B 0,C 180,E1 9507.843,E2 9507.843} C_VEL
LIN {X 0,Y 244.136,Z 731.046,A -85,B 0,C 180,E1 9505.404,E2 9505.404} C_VEL
LIN {X 0,Y 234.176,Z 746.412,A -85,B 0,C 180,E1 9502.574,E2 9502.574} C_VEL
LIN {X 0,Y 224.191,Z 760.266,A -85,B 0,C 180,E1 9499.302,E2 9499.302} C_VEL
LIN {X 0,Y 214.412,Z 772.729,A -85,B 0,C 180,E1 9495.517,E2 9495.517} C_VEL
LIN {X 0,Y 204.639,Z 784.419,A -85,B 0,C 180,E1 9490.897,E2 9490.897} C_VEL
LIN {X 0,Y 196.206,Z 794.078,A -85,B 0,C 180,E1 9485.875,E2 9485.875} C_VEL
LIN {X 0,Y 188.932,Z 802.31,A -85,B 0,C 180,E1 9480.181,E2 9480.181} C_VEL
LIN {X 0,Y 183.148,Z 808.941,A -85,B 0,C 180,E1 9473.827,E2 9473.827} C_VEL
LIN {X 0,Y 179.282,Z 813.77,A -85,B 0,C 180,E1 9467.192,E2 9467.192} C_VEL
LIN {X 0,Y 177.197,Z 816.943,A -85,B 0,C 180,E1 9460.402,E2 9460.402} C_VEL
LIN {X 0,Y 176.465,Z 818.477,A -85,B 0,C 180,E1 9454.224,E2 9454.224} C_VEL
LIN {X 0,Y 176.37,Z 818.696,A -85,B 0,C 180,E1 9448.376,E2 9448.376} C_VEL
LIN {X 0,Y 176.771,Z 817.818,A -85,B 0,C 180,E1 9442.198,E2 9442.198} C_VEL
LIN {X 0,Y 178.169,Z 815.404,A -85,B 0,C 180,E1 9435.705,E2 9435.705} C_VEL
LIN {X 0,Y 181.403,Z 811.078,A -85,B 0,C 180,E1 9428.668,E2 9428.668} C_VEL
LIN {X 0,Y 186.427,Z 805.167,A -85,B 0,C 180,E1 9422.187,E2 9422.187} C_VEL
LIN {X 0,Y 193.014,Z 797.799,A -85,B 0,C 180,E1 9416.34,E2 9416.34} C_VEL
LIN {X 0,Y 201.645,Z 788.048,A -85,B 0,C 180,E1 9410.673,E2 9410.673} C_VEL
LIN {X 0,Y 210.551,Z 777.57,A -85,B 0,C 180,E1 9406.108,E2 9406.108} C_VEL
LIN {X 0,Y 220.518,Z 765.194,A -85,B 0,C 180,E1 9401.963,E2 9401.963} C_VEL
LIN {X 0,Y 230.846,Z 751.31,A -85,B 0,C 180,E1 9398.377,E2 9398.377} C_VEL
LIN {X 0,Y 240.967,Z 736.387,A -85,B 0,C 180,E1 9395.381,E2 9395.381} C_VEL
LIN {X 0,Y 250.781,Z 720.142,A -85,B 0,C 180,E1 9392.836,E2 9392.836} C_VEL
LIN {X 0,Y 259.56,Z 703.613,A -85,B 0,C 180,E1 9390.795,E2 9390.795} C_VEL
LIN {X 0,Y 268.075,Z 685.252,A -85,B 0,C 180,E1 9389.004,E2 9389.004} C_VEL
LIN {X 0,Y 275.289,Z 667.039,A -85,B 0,C 180,E1 9387.601,E2 9387.601} C_VEL
LIN {X 0,Y 281.862,Z 646.773,A -85,B 0,C 180,E1 9386.405,E2 9386.405} C_VEL
LIN {X 0,Y 287.054,Z 626.277,A -85,B 0,C 180,E1 9385.501,E2 9385.501} C_VEL
LIN {X 0,Y 291.037,Z 604.846,A -85,B 0,C 180,E1 9384.826,E2 9384.826} C_VEL
LIN {X 0,Y 293.813,Z 580.425,A -85,B 0,C 180,E1 9384.283,E2 9384.283} C_VEL
LIN {X 0,Y 304.982,Z 454.841,A -85,B 0,C 180,E1 9381.796,E2 9381.796} C_VEL
LIN {X 0,Y 301.25,Z 446.677,A -85,B 0,C 180,E1 9379.032,E2 9379.032} C_VEL
LIN {X 0,Y 297.914,Z 439.839,A -85,B 0,C 180,E1 9376.075,E2 9376.075} C_VEL
LIN {X 0,Y 295.788,Z 435.718,A -85,B 0,C 180,E1 9373.787,E2 9373.787} C_VEL
LIN {X 0,Y 294.274,Z 432.633,A -85,B 0,C 180,E1 9371.763,E2 9371.763} C_VEL
LIN {X 0,Y 292.797,Z 429.694,A -85,B 0,C 180,E1 9369.236,E2 9369.236} C_VEL
LIN {X 0,Y 291.284,Z 426.041,A -85,B 0,C 180,E1 9364.134,E2 9364.134} C_VEL
LIN {X 0,Y 291.551,Z 426.128,A -85,B 0,C 180,E1 9359.411,E2 9359.411} C_VEL
LIN {X 0,Y 292.669,Z 428.684,A -85,B 0,C 180,E1 9355.97,E2 9355.97} C_VEL
LIN {X 0,Y 293.219,Z 430.558,A -85,B 0,C 180,E1 9354.727,E2 9354.727} C_VEL
LIN {X 0,Y 294.022,Z 435.945,A -85,B 0,C 180,E1 9352.822,E2 9352.822} C_VEL
LIN {X 0,Y 295.341,Z 442.859,A -85,B 0,C 180,E1 9350.565,E2 9350.565} C_VEL
LIN {X 0,Y 296.023,Z 444.519,A -85,B 0,C 180,E1 9349.765,E2 9349.765} C_VEL
LIN {X 0,Y 298.848,Z 449.865,A -85,B 0,C 180,E1 9347.047,E2 9347.047} C_VEL
LIN {X 0,Y 302.677,Z 457.738,A -85,B 0,C 180,E1 9343.989,E2 9343.989} C_VEL
LIN {X 0,Y 302.886,Z 458.631,A -85,B 0,C 180,E1 9343.803,E2 9343.803} C_VEL
LIN {X 0,Y 288.854,Z 601.913,A -85,B 0,C 180,E1 9340.891,E2 9340.891} C_VEL
LIN {X 0,Y 284.976,Z 623.979,A -85,B 0,C 180,E1 9340.282,E2 9340.282} C_VEL
LIN {X 0,Y 279.696,Z 645.376,A -85,B 0,C 180,E1 9339.484,E2 9339.484} C_VEL
LIN {X 0,Y 273.109,Z 666.357,A -85,B 0,C 180,E1 9338.415,E2 9338.415} C_VEL
LIN {X 0,Y 265.841,Z 685.527,A -85,B 0,C 180,E1 9337.138,E2 9337.138} C_VEL
LIN {X 0,Y 257.139,Z 704.754,A -85,B 0,C 180,E1 9335.486,E2 9335.486} C_VEL
LIN {X 0,Y 247.561,Z 723.186,A -85,B 0,C 180,E1 9333.454,E2 9333.454} C_VEL
LIN {X 0,Y 237.443,Z 740.435,A -85,B 0,C 180,E1 9331.037,E2 9331.037} C_VEL
LIN {X 0,Y 227.088,Z 756.393,A -85,B 0,C 180,E1 9328.184,E2 9328.184} C_VEL
LIN {X 0,Y 216.175,Z 771.6,A -85,B 0,C 180,E1 9324.68,E2 9324.68} C_VEL
LIN {X 0,Y 205.676,Z 785.255,A -85,B 0,C 180,E1 9320.618,E2 9320.618} C_VEL
LIN {X 0,Y 195.491,Z 797.894,A -85,B 0,C 180,E1 9315.727,E2 9315.727} C_VEL
LIN {X 0,Y 186.783,Z 808.53,A -85,B 0,C 180,E1 9310.368,E2 9310.368} C_VEL
LIN {X 0,Y 179.378,Z 817.668,A -85,B 0,C 180,E1 9304.261,E2 9304.261} C_VEL
LIN {X 0,Y 173.834,Z 825.097,A -85,B 0,C 180,E1 9297.654,E2 9297.654} C_VEL
LIN {X 0,Y 170.216,Z 830.927,A -85,B 0,C 180,E1 9290.636,E2 9290.636} C_VEL
LIN {X 0,Y 168.57,Z 834.724,A -85,B 0,C 180,E1 9284.074,E2 9284.074} C_VEL
LIN {X 0,Y 168.182,Z 837.189,A -85,B 0,C 180,E1 9277.172,E2 9277.172} C_VEL
LIN {X 0,Y 168.279,Z 837.996,A -85,B 0,C 180,E1 9272.043,E2 9272.043} C_VEL
LIN {X 0,Y 168.264,Z 837.941,A -85,B 0,C 180,E1 9267.275,E2 9267.275} C_VEL
LIN {X 0,Y 168.178,Z 836.862,A -85,B 0,C 180,E1 9261.453,E2 9261.453} C_VEL
LIN {X 0,Y 168.734,Z 834.173,A -85,B 0,C 180,E1 9254.887,E2 9254.887} C_VEL
LIN {X 0,Y 170.905,Z 829.643,A -85,B 0,C 180,E1 9247.65,E2 9247.65} C_VEL
LIN {X 0,Y 175.083,Z 823.337,A -85,B 0,C 180,E1 9240.586,E2 9240.586} C_VEL
LIN {X 0,Y 181.047,Z 815.465,A -85,B 0,C 180,E1 9234.17,E2 9234.17} C_VEL
LIN {X 0,Y 188.909,Z 805.78,A -85,B 0,C 180,E1 9228.174,E2 9228.174} C_VEL
LIN {X 0,Y 198.025,Z 794.708,A -85,B 0,C 180,E1 9222.937,E2 9222.937} C_VEL
LIN {X 0,Y 208.464,Z 781.653,A -85,B 0,C 180,E1 9218.222,E2 9218.222} C_VEL
LIN {X 0,Y 219.096,Z 767.46,A -85,B 0,C 180,E1 9214.312,E2 9214.312} C_VEL
LIN {X 0,Y 229.812,Z 752.056,A -85,B 0,C 180,E1 9211.01,E2 9211.01} C_VEL
LIN {X 0,Y 240.491,Z 735.201,A -85,B 0,C 180,E1 9208.191,E2 9208.191} C_VEL
LIN {X 0,Y 250.581,Z 717.449,A -85,B 0,C 180,E1 9205.874,E2 9205.874} C_VEL
LIN {X 0,Y 259.873,Z 698.684,A -85,B 0,C 180,E1 9203.971,E2 9203.971} C_VEL
LIN {X 0,Y 267.846,Z 680.035,A -85,B 0,C 180,E1 9202.49,E2 9202.49} C_VEL
LIN {X 0,Y 275.147,Z 659.876,A -85,B 0,C 180,E1 9201.24,E2 9201.24} C_VEL
LIN {X 0,Y 281.357,Z 638.826,A -85,B 0,C 180,E1 9200.257,E2 9200.257} C_VEL
LIN {X 0,Y 286.185,Z 617.107,A -85,B 0,C 180,E1 9199.528,E2 9199.528} C_VEL
LIN {X 0,Y 289.444,Z 595.253,A -85,B 0,C 180,E1 9198.973,E2 9198.973} C_VEL
LIN {X 0,Y 302.688,Z 458.042,A -85,B 0,C 180,E1 9196.158,E2 9196.158} C_VEL
LIN {X 0,Y 298.869,Z 450.155,A -85,B 0,C 180,E1 9193.149,E2 9193.149} C_VEL
LIN {X 0,Y 295.986,Z 444.625,A -85,B 0,C 180,E1 9190.412,E2 9190.412} C_VEL
LIN {X 0,Y 294.079,Z 441.082,A -85,B 0,C 180,E1 9188.209,E2 9188.209} C_VEL
LIN {X 0,Y 292.366,Z 437.787,A -85,B 0,C 180,E1 9185.691,E2 9185.691} C_VEL
LIN {X 0,Y 290.37,Z 433.935,A -85,B 0,C 180,E1 9180.789,E2 9180.789} C_VEL
LIN {X 0,Y 290.021,Z 433.788,A -85,B 0,C 180,E1 9176.046,E2 9176.046} C_VEL
LIN {X 0,Y 290.292,Z 434.605,A -85,B 0,C 180,E1 9174.267,E2 9174.267} C_VEL
LIN {X 0,Y 291.993,Z 438.415,A -85,B 0,C 180,E1 9169.842,E2 9169.842} C_VEL
LIN {X 0,Y 293.768,Z 442.12,A -85,B 0,C 180,E1 9167.118,E2 9167.118} C_VEL
LIN {X 0,Y 296.075,Z 446.883,A -85,B 0,C 180,E1 9164.426,E2 9164.426} C_VEL
LIN {X 0,Y 299.327,Z 453.827,A -85,B 0,C 180,E1 9161.397,E2 9161.397} C_VEL
LIN {X 0,Y 301.811,Z 459.604,A -85,B 0,C 180,E1 9159.417,E2 9159.417} C_VEL
LIN {X 0,Y 288.8,Z 598.714,A -85,B 0,C 180,E1 9156.695,E2 9156.695} C_VEL
LIN {X 0,Y 285.13,Z 620.197,A -85,B 0,C 180,E1 9156.093,E2 9156.093} C_VEL
LIN {X 0,Y 280.34,Z 640.174,A -85,B 0,C 180,E1 9155.308,E2 9155.308} C_VEL
LIN {X 0,Y 274.177,Z 660.226,A -85,B 0,C 180,E1 9154.253,E2 9154.253} C_VEL
LIN {X 0,Y 267.139,Z 678.981,A -85,B 0,C 180,E1 9152.97,E2 9152.97} C_VEL
LIN {X 0,Y 258.696,Z 697.645,A -85,B 0,C 180,E1 9151.322,E2 9151.322} C_VEL
LIN {X 0,Y 249.743,Z 714.709,A -85,B 0,C 180,E1 9149.4,E2 9149.4} C_VEL
LIN {X 0,Y 239.664,Z 731.577,A -85,B 0,C 180,E1 9146.985,E2 9146.985} C_VEL
LIN {X 0,Y 230.041,Z 745.999,A -85,B 0,C 180,E1 9144.366,E2 9144.366} C_VEL
LIN {X 0,Y 219.369,Z 760.294,A -85,B 0,C 180,E1 9141.024,E2 9141.024} C_VEL
LIN {X 0,Y 209.225,Z 772.731,A -85,B 0,C 180,E1 9137.265,E2 9137.265} C_VEL
LIN {X 0,Y 199.093,Z 784.332,A -85,B 0,C 180,E1 9132.685,E2 9132.685} C_VEL
LIN {X 0,Y 190.127,Z 794.098,A -85,B 0,C 180,E1 9127.591,E2 9127.591} C_VEL
LIN {X 0,Y 182.31,Z 802.387,A -85,B 0,C 180,E1 9121.768,E2 9121.768} C_VEL
LIN {X 0,Y 176.267,Z 808.823,A -85,B 0,C 180,E1 9115.537,E2 9115.537} C_VEL
LIN {X 0,Y 171.786,Z 813.97,A -85,B 0,C 180,E1 9108.426,E2 9108.426} C_VEL
LIN {X 0,Y 169.372,Z 817.289,A -85,B 0,C 180,E1 9101.233,E2 9101.233} C_VEL
LIN {X 0,Y 168.506,Z 818.863,A -85,B 0,C 180,E1 9094.765,E2 9094.765} C_VEL
LIN {X 0,Y 168.381,Z 819.165,A -85,B 0,C 180,E1 9088.639,E2 9088.639} C_VEL
LIN {X 0,Y 168.739,Z 818.392,A -85,B 0,C 180,E1 9082.51,E2 9082.51} C_VEL
LIN {X 0,Y 170.148,Z 816.154,A -85,B 0,C 180,E1 9075.712,E2 9075.712} C_VEL
LIN {X 0,Y 173.284,Z 812.254,A -85,B 0,C 180,E1 9068.685,E2 9068.685} C_VEL
LIN {X 0,Y 178.401,Z 806.632,A -85,B 0,C 180,E1 9061.916,E2 9061.916} C_VEL
LIN {X 0,Y 185.531,Z 799.057,A -85,B 0,C 180,E1 9055.539,E2 9055.539} C_VEL
LIN {X 0,Y 193.626,Z 790.407,A -85,B 0,C 180,E1 9050.186,E2 9050.186} C_VEL
LIN {X 0,Y 203.165,Z 779.887,A -85,B 0,C 180,E1 9045.272,E2 9045.272} C_VEL
LIN {X 0,Y 213.395,Z 767.927,A -85,B 0,C 180,E1 9041.032,E2 9041.032} C_VEL
LIN {X 0,Y 224.019,Z 754.447,A -85,B 0,C 180,E1 9037.374,E2 9037.374} C_VEL
LIN {X 0,Y 234.668,Z 739.452,A -85,B 0,C 180,E1 9034.253,E2 9034.253} C_VEL
LIN {X 0,Y 244.53,Z 723.971,A -85,B 0,C 180,E1 9031.738,E2 9031.738} C_VEL
LIN {X 0,Y 254.062,Z 707.098,A -85,B 0,C 180,E1 9029.574,E2 9029.574} C_VEL
LIN {X 0,Y 262.751,Z 689.491,A -85,B 0,C 180,E1 9027.796,E2 9027.796} C_VEL
LIN {X 0,Y 270.448,Z 670.99,A -85,B 0,C 180,E1 9026.337,E2 9026.337} C_VEL
LIN {X 0,Y 277.221,Z 651.449,A -85,B 0,C 180,E1 9025.141,E2 9025.141} C_VEL
LIN {X 0,Y 282.921,Z 630.853,A -85,B 0,C 180,E1 9024.188,E2 9024.188} C_VEL
LIN {X 0,Y 287.255,Z 610.009,A -85,B 0,C 180,E1 9023.487,E2 9023.487} C_VEL
LIN {X 0,Y 290.197,Z 587.919,A -85,B 0,C 180,E1 9022.969,E2 9022.969} C_VEL
LIN {X 0,Y 301.96,Z 459.498,A -85,B 0,C 180,E1 9020.447,E2 9020.447} C_VEL
LIN {X 0,Y 298.474,Z 451.727,A -85,B 0,C 180,E1 9017.598,E2 9017.598} C_VEL
LIN {X 0,Y 295.312,Z 444.935,A -85,B 0,C 180,E1 9014.41,E2 9014.41} C_VEL
LIN {X 0,Y 293.101,Z 440.447,A -85,B 0,C 180,E1 9011.512,E2 9011.512} C_VEL
LIN {X 0,Y 291.723,Z 437.579,A -85,B 0,C 180,E1 9009.072,E2 9009.072} C_VEL
LIN {X 0,Y 290.311,Z 433.987,A -85,B 0,C 180,E1 9004.148,E2 9004.148} C_VEL
LIN {X 0,Y 290.566,Z 434.075,A -85,B 0,C 180,E1 8999.409,E2 8999.409} C_VEL
LIN {X 0,Y 292.939,Z 438.619,A -85,B 0,C 180,E1 8993.73,E2 8993.73} C_VEL
LIN {X 0,Y 295.32,Z 443.156,A -85,B 0,C 180,E1 8990.549,E2 8990.549} C_VEL
LIN {X 0,Y 296.023,Z 444.519,A -85,B 0,C 180,E1 8989.765,E2 8989.765} C_VEL
LIN {X 0,Y 296.729,Z 447.072,A -85,B 0,C 180,E1 8988.904,E2 8988.904} C_VEL
LIN {X 0,Y 298.105,Z 458.569,A -85,B 0,C 180,E1 8986.779,E2 8986.779} C_VEL
LIN {X 0,Y 298.603,Z 460.189,A -85,B 0,C 180,E1 8986.297,E2 8986.297} C_VEL
LIN {X 0,Y 299.955,Z 463.363,A -85,B 0,C 180,E1 8985.161,E2 8985.161} C_VEL
LIN {X 0,Y 286.061,Z 601.776,A -85,B 0,C 180,E1 8982.391,E2 8982.391} C_VEL
LIN {X 0,Y 282.107,Z 623.842,A -85,B 0,C 180,E1 8981.797,E2 8981.797} C_VEL
LIN {X 0,Y 276.73,Z 645.196,A -85,B 0,C 180,E1 8981.024,E2 8981.024} C_VEL
LIN {X 0,Y 269.868,Z 666.532,A -85,B 0,C 180,E1 8979.964,E2 8979.964} C_VEL
LIN {X 0,Y 262.367,Z 685.777,A -85,B 0,C 180,E1 8978.708,E2 8978.708} C_VEL
LIN {X 0,Y 253.053,Z 705.763,A -85,B 0,C 180,E1 8977.014,E2 8977.014} C_VEL
LIN {X 0,Y 243.225,Z 723.967,A -85,B 0,C 180,E1 8975.015,E2 8975.015} C_VEL
LIN {X 0,Y 232.237,Z 741.917,A -85,B 0,C 180,E1 8972.483,E2 8972.483} C_VEL
LIN {X 0,Y 221.425,Z 757.797,A -85,B 0,C 180,E1 8969.593,E2 8969.593} C_VEL
LIN {X 0,Y 209.905,Z 773.186,A -85,B 0,C 180,E1 8965.976,E2 8965.976} C_VEL
LIN {X 0,Y 198.718,Z 786.938,A -85,B 0,C 180,E1 8961.711,E2 8961.711} C_VEL
LIN {X 0,Y 188.341,Z 799.045,A -85,B 0,C 180,E1 8956.778,E2 8956.778} C_VEL
LIN {X 0,Y 178.77,Z 809.982,A -85,B 0,C 180,E1 8950.871,E2 8950.871} C_VEL
LIN {X 0,Y 171.211,Z 818.83,A -85,B 0,C 180,E1 8944.504,E2 8944.504} C_VEL
LIN {X 0,Y 165.417,Z 826.174,A -85,B 0,C 180,E1 8937.311,E2 8937.311} C_VEL
LIN {X 0,Y 162.007,Z 831.36,A -85,B 0,C 180,E1 8930.219,E2 8930.219} C_VEL
LIN {X 0,Y 160.43,Z 835.056,A -85,B 0,C 180,E1 8922.965,E2 8922.965} C_VEL
LIN {X 0,Y 160.197,Z 836.966,A -85,B 0,C 180,E1 8916.45,E2 8916.45} C_VEL
LIN {X 0,Y 160.312,Z 837.647,A -85,B 0,C 180,E1 8910.715,E2 8910.715} C_VEL
LIN {X 0,Y 160.222,Z 837.257,A -85,B 0,C 180,E1 8904.988,E2 8904.988} C_VEL
LIN {X 0,Y 160.279,Z 835.666,A -85,B 0,C 180,E1 8898.85,E2 8898.85} C_VEL
LIN {X 0,Y 161.451,Z 832.439,A -85,B 0,C 180,E1 8891.589,E2 8891.589} C_VEL
LIN {X 0,Y 164.39,Z 827.542,A -85,B 0,C 180,E1 8884.416,E2 8884.416} C_VEL
LIN {X 0,Y 169.623,Z 820.642,A -85,B 0,C 180,E1 8877.161,E2 8877.161} C_VEL
LIN {X 0,Y 176.69,Z 812.31,A -85,B 0,C 180,E1 8870.671,E2 8870.671} C_VEL
LIN {X 0,Y 185.675,Z 802.072,A -85,B 0,C 180,E1 8864.7,E2 8864.7} C_VEL
LIN {X 0,Y 195.806,Z 790.263,A -85,B 0,C 180,E1 8859.553,E2 8859.553} C_VEL
LIN {X 0,Y 206.714,Z 776.978,A -85,B 0,C 180,E1 8855.141,E2 8855.141} C_VEL
LIN {X 0,Y 217.93,Z 762.383,A -85,B 0,C 180,E1 8851.423,E2 8851.423} C_VEL
LIN {X 0,Y 228.925,Z 746.821,A -85,B 0,C 180,E1 8848.351,E2 8848.351} C_VEL
LIN {X 0,Y 239.376,Z 730.284,A -85,B 0,C 180,E1 8845.828,E2 8845.828} C_VEL
LIN {X 0,Y 249.467,Z 712.342,A -85,B 0,C 180,E1 8843.681,E2 8843.681} C_VEL
LIN {X 0,Y 258.685,Z 693.648,A -85,B 0,C 180,E1 8841.934,E2 8841.934} C_VEL
LIN {X 0,Y 266.889,Z 674.238,A -85,B 0,C 180,E1 8840.518,E2 8840.518} C_VEL
LIN {X 0,Y 273.885,Z 654.133,A -85,B 0,C 180,E1 8839.403,E2 8839.403} C_VEL
LIN {X 0,Y 279.795,Z 633.049,A -85,B 0,C 180,E1 8838.528,E2 8838.528} C_VEL
LIN {X 0,Y 284.328,Z 611.476,A -85,B 0,C 180,E1 8837.87,E2 8837.87} C_VEL
LIN {X 0,Y 287.35,Z 589.153,A -85,B 0,C 180,E1 8837.346,E2 8837.346} C_VEL
LIN {X 0,Y 299.774,Z 463.048,A -85,B 0,C 180,E1 8834.832,E2 8834.832} C_VEL
LIN {X 0,Y 296.476,Z 455.999,A -85,B 0,C 180,E1 8831.97,E2 8831.97} C_VEL
LIN {X 0,Y 293.686,Z 450.489,A -85,B 0,C 180,E1 8829.01,E2 8829.01} C_VEL
LIN {X 0,Y 291.136,Z 445.506,A -85,B 0,C 180,E1 8825.32,E2 8825.32} C_VEL
LIN {X 0,Y 289.337,Z 441.837,A -85,B 0,C 180,E1 8820.594,E2 8820.594} C_VEL
LIN {X 0,Y 289.073,Z 441.757,A -85,B 0,C 180,E1 8815.834,E2 8815.834} C_VEL
LIN {X 0,Y 289.542,Z 443.483,A -85,B 0,C 180,E1 8813.257,E2 8813.257} C_VEL
LIN {X 0,Y 290.857,Z 446.246,A -85,B 0,C 180,E1 8810.102,E2 8810.102} C_VEL
LIN {X 0,Y 292.495,Z 449.843,A -85,B 0,C 180,E1 8807.463,E2 8807.463} C_VEL
LIN {X 0,Y 294.719,Z 454.636,A -85,B 0,C 180,E1 8804.756,E2 8804.756} C_VEL
LIN {X 0,Y 297.93,Z 461.812,A -85,B 0,C 180,E1 8801.661,E2 8801.661} C_VEL
LIN {X 0,Y 298.934,Z 464.55,A -85,B 0,C 180,E1 8800.783,E2 8800.783} C_VEL
LIN {X 0,Y 285.99,Z 598.881,A -85,B 0,C 180,E1 8798.189,E2 8798.189} C_VEL
LIN {X 0,Y 282.222,Z 620.441,A -85,B 0,C 180,E1 8797.599,E2 8797.599} C_VEL
LIN {X 0,Y 277.319,Z 640.409,A -85,B 0,C 180,E1 8796.833,E2 8796.833} C_VEL
LIN {X 0,Y 271.074,Z 660.295,A -85,B 0,C 180,E1 8795.813,E2 8795.813} C_VEL
LIN {X 0,Y 264.008,Z 678.727,A -85,B 0,C 180,E1 8794.586,E2 8794.586} C_VEL
LIN {X 0,Y 255.473,Z 697.211,A -85,B 0,C 180,E1 8792.999,E2 8792.999} C_VEL
LIN {X 0,Y 246.169,Z 714.571,A -85,B 0,C 180,E1 8791.096,E2 8791.096} C_VEL
LIN {X 0,Y 236.111,Z 731.018,A -85,B 0,C 180,E1 8788.802,E2 8788.802} C_VEL
LIN {X 0,Y 225.397,Z 746.57,A -85,B 0,C 180,E1 8786.017,E2 8786.017} C_VEL
LIN {X 0,Y 214.197,Z 761.028,A -85,B 0,C 180,E1 8782.638,E2 8782.638} C_VEL
LIN {X 0,Y 203.403,Z 773.69,A -85,B 0,C 180,E1 8778.77,E2 8778.77} C_VEL
LIN {X 0,Y 192.682,Z 785.357,A -85,B 0,C 180,E1 8774.053,E2 8774.053} C_VEL
LIN {X 0,Y 183.308,Z 795.001,A -85,B 0,C 180,E1 8768.848,E2 8768.848} C_VEL
LIN {X 0,Y 175.1,Z 803.23,A -85,B 0,C 180,E1 8762.851,E2 8762.851} C_VEL
LIN {X 0,Y 168.452,Z 809.857,A -85,B 0,C 180,E1 8756.054,E2 8756.054} C_VEL
LIN {X 0,Y 163.919,Z 814.679,A -85,B 0,C 180,E1 8748.861,E2 8748.861} C_VEL
LIN {X 0,Y 161.412,Z 817.845,A -85,B 0,C 180,E1 8741.433,E2 8741.433} C_VEL
LIN {X 0,Y 160.512,Z 819.376,A -85,B 0,C 180,E1 8734.645,E2 8734.645} C_VEL
LIN {X 0,Y 160.396,Z 819.592,A -85,B 0,C 180,E1 8728.214,E2 8728.214} C_VEL
LIN {X 0,Y 160.84,Z 818.779,A -85,B 0,C 180,E1 8721.78,E2 8721.78} C_VEL
LIN {X 0,Y 162.465,Z 816.456,A -85,B 0,C 180,E1 8714.655,E2 8714.655} C_VEL
LIN {X 0,Y 166.202,Z 812.227,A -85,B 0,C 180,E1 8706.982,E2 8706.982} C_VEL
LIN {X 0,Y 171.921,Z 806.418,A -85,B 0,C 180,E1 8699.99,E2 8699.99} C_VEL
LIN {X 0,Y 179.728,Z 798.72,A -85,B 0,C 180,E1 8693.47,E2 8693.47} C_VEL
LIN {X 0,Y 188.965,Z 789.375,A -85,B 0,C 180,E1 8687.781,E2 8687.781} C_VEL
LIN {X 0,Y 198.626,Z 779.122,A -85,B 0,C 180,E1 8683.123,E2 8683.123} C_VEL
LIN {X 0,Y 209.425,Z 766.906,A -85,B 0,C 180,E1 8678.905,E2 8678.905} C_VEL
LIN {X 0,Y 219.85,Z 754.118,A -85,B 0,C 180,E1 8675.506,E2 8675.506} C_VEL
LIN {X 0,Y 231.31,Z 738.468,A -85,B 0,C 180,E1 8672.324,E2 8672.324} C_VEL
LIN {X 0,Y 241.521,Z 722.717,A -85,B 0,C 180,E1 8669.857,E2 8669.857} C_VEL
LIN {X 0,Y 251.411,Z 705.409,A -85,B 0,C 180,E1 8667.731,E2 8667.731} C_VEL
LIN {X 0,Y 260.319,Z 687.449,A -85,B 0,C 180,E1 8666.007,E2 8666.007} C_VEL
LIN {X 0,Y 268.278,Z 668.546,A -85,B 0,C 180,E1 8664.584,E2 8664.584} C_VEL
LIN {X 0,Y 275.156,Z 648.472,A -85,B 0,C 180,E1 8663.436,E2 8663.436} C_VEL
LIN {X 0,Y 280.704,Z 627.962,A -85,B 0,C 180,E1 8662.555,E2 8662.555} C_VEL
LIN {X 0,Y 285.108,Z 605.741,A -85,B 0,C 180,E1 8661.875,E2 8661.875} C_VEL
LIN {X 0,Y 287.961,Z 582.541,A -85,B 0,C 180,E1 8661.37,E2 8661.37} C_VEL
LIN {X 0,Y 299.098,Z 464.293,A -85,B 0,C 180,E1 8659.073,E2 8659.073} C_VEL
LIN {X 0,Y 295.408,Z 455.833,A -85,B 0,C 180,E1 8655.66,E2 8655.66} C_VEL
LIN {X 0,Y 293.2,Z 451.143,A -85,B 0,C 180,E1 8653.108,E2 8653.108} C_VEL
LIN {X 0,Y 291.739,Z 447.917,A -85,B 0,C 180,E1 8650.966,E2 8650.966} C_VEL
LIN {X 0,Y 290.557,Z 445.318,A -85,B 0,C 180,E1 8648.709,E2 8648.709} C_VEL
LIN {X 0,Y 289.313,Z 441.904,A -85,B 0,C 180,E1 8643.964,E2 8643.964} C_VEL
LIN {X 0,Y 289.581,Z 442.025,A -85,B 0,C 180,E1 8639.407,E2 8639.407} C_VEL
LIN {X 0,Y 291.754,Z 446.442,A -85,B 0,C 180,E1 8634.001,E2 8634.001} C_VEL
LIN {X 0,Y 293.971,Z 450.855,A -85,B 0,C 180,E1 8630.9,E2 8630.9} C_VEL
LIN {X 0,Y 296.873,Z 456.527,A -85,B 0,C 180,E1 8627.849,E2 8627.849} C_VEL
LIN {X 0,Y 298.603,Z 460.189,A -85,B 0,C 180,E1 8626.297,E2 8626.297} C_VEL
LIN {X 0,Y 298.876,Z 462.06,A -85,B 0,C 180,E1 8625.954,E2 8625.954} C_VEL
LIN {X 0,Y 298.651,Z 466.09,A -85,B 0,C 180,E1 8625.757,E2 8625.757} C_VEL
LIN {X 0,Y 297.656,Z 472.141,A -85,B 0,C 180,E1 8625.891,E2 8625.891} C_VEL
LIN {X 0,Y 295.908,Z 481.417,A -85,B 0,C 180,E1 8626.248,E2 8626.248} C_VEL
LIN {X 0,Y 295.583,Z 483.996,A -85,B 0,C 180,E1 8626.24,E2 8626.24} C_VEL
LIN {X 0,Y 283.455,Z 601.742,A -85,B 0,C 180,E1 8623.916,E2 8623.916} C_VEL
LIN {X 0,Y 279.406,Z 623.866,A -85,B 0,C 180,E1 8623.337,E2 8623.337} C_VEL
LIN {X 0,Y 274.14,Z 644.427,A -85,B 0,C 180,E1 8622.62,E2 8622.62} C_VEL
LIN {X 0,Y 267.551,Z 664.783,A -85,B 0,C 180,E1 8621.657,E2 8621.657} C_VEL
LIN {X 0,Y 259.517,Z 685.088,A -85,B 0,C 180,E1 8620.386,E2 8620.386} C_VEL
LIN {X 0,Y 250.487,Z 704.081,A -85,B 0,C 180,E1 8618.837,E2 8618.837} C_VEL
LIN {X 0,Y 240.265,Z 722.704,A -85,B 0,C 180,E1 8616.877,E2 8616.877} C_VEL
LIN {X 0,Y 229.309,Z 740.241,A -85,B 0,C 180,E1 8614.496,E2 8614.496} C_VEL
LIN {X 0,Y 218.083,Z 756.333,A -85,B 0,C 180,E1 8611.672,E2 8611.672} C_VEL
LIN {X 0,Y 206.059,Z 771.818,A -85,B 0,C 180,E1 8608.117,E2 8608.117} C_VEL
LIN {X 0,Y 194.914,Z 784.996,A -85,B 0,C 180,E1 8604.142,E2 8604.142} C_VEL
LIN {X 0,Y 183.688,Z 797.531,A -85,B 0,C 180,E1 8599.165,E2 8599.165} C_VEL
LIN {X 0,Y 173.874,Z 808.133,A -85,B 0,C 180,E1 8593.569,E2 8593.569} C_VEL
LIN {X 0,Y 165.409,Z 817.266,A -85,B 0,C 180,E1 8587.07,E2 8587.07} C_VEL
LIN {X 0,Y 158.883,Z 824.71,A -85,B 0,C 180,E1 8579.811,E2 8579.811} C_VEL
LIN {X 0,Y 154.459,Z 830.675,A -85,B 0,C 180,E1 8571.652,E2 8571.652} C_VEL
LIN {X 0,Y 152.55,Z 834.473,A -85,B 0,C 180,E1 8564.034,E2 8564.034} C_VEL
LIN {X 0,Y 152.199,Z 836.439,A -85,B 0,C 180,E1 8557.17,E2 8557.17} C_VEL
LIN {X 0,Y 152.313,Z 837.15,A -85,B 0,C 180,E1 8551.505,E2 8551.505} C_VEL
LIN {X 0,Y 152.25,Z 836.961,A -85,B 0,C 180,E1 8545.857,E2 8545.857} C_VEL
LIN {X 0,Y 152.272,Z 835.461,A -85,B 0,C 180,E1 8539.023,E2 8539.023} C_VEL
LIN {X 0,Y 153.367,Z 832.555,A -85,B 0,C 180,E1 8531.765,E2 8531.765} C_VEL
LIN {X 0,Y 156.345,Z 827.894,A -85,B 0,C 180,E1 8524.224,E2 8524.224} C_VEL
LIN {X 0,Y 161.739,Z 821.294,A -85,B 0,C 180,E1 8516.621,E2 8516.621} C_VEL
LIN {X 0,Y 169.424,Z 812.851,A -85,B 0,C 180,E1 8509.578,E2 8509.578} C_VEL
LIN {X 0,Y 178.868,Z 802.668,A -85,B 0,C 180,E1 8503.392,E2 8503.392} C_VEL
LIN {X 0,Y 188.824,Z 791.75,A -85,B 0,C 180,E1 8498.403,E2 8498.403} C_VEL
LIN {X 0,Y 200.03,Z 778.915,A -85,B 0,C 180,E1 8493.928,E2 8493.928} C_VEL
LIN {X 0,Y 211.6,Z 764.698,A -85,B 0,C 180,E1 8490.152,E2 8490.152} C_VEL
LIN {X 0,Y 223.24,Z 748.911,A -85,B 0,C 180,E1 8486.967,E2 8486.967} C_VEL
LIN {X 0,Y 234.337,Z 732.202,A -85,B 0,C 180,E1 8484.367,E2 8484.367} C_VEL
LIN {X 0,Y 245.074,Z 713.97,A -85,B 0,C 180,E1 8482.166,E2 8482.166} C_VEL
LIN {X 0,Y 254.502,Z 695.699,A -85,B 0,C 180,E1 8480.452,E2 8480.452} C_VEL
LIN {X 0,Y 263.294,Z 675.54,A -85,B 0,C 180,E1 8478.994,E2 8478.994} C_VEL
LIN {X 0,Y 270.541,Z 655.519,A -85,B 0,C 180,E1 8477.892,E2 8477.892} C_VEL
LIN {X 0,Y 276.844,Z 633.852,A -85,B 0,C 180,E1 8477.005,E2 8477.005} C_VEL
LIN {X 0,Y 281.486,Z 612.618,A -85,B 0,C 180,E1 8476.367,E2 8476.367} C_VEL
LIN {X 0,Y 284.67,Z 590.099,A -85,B 0,C 180,E1 8475.845,E2 8475.845} C_VEL
LIN {X 0,Y 296.963,Z 468.005,A -85,B 0,C 180,E1 8473.433,E2 8473.433} C_VEL
LIN {X 0,Y 293.669,Z 460.797,A -85,B 0,C 180,E1 8470.197,E2 8470.197} C_VEL
LIN {X 0,Y 291.404,Z 456.313,A -85,B 0,C 180,E1 8467.392,E2 8467.392} C_VEL
LIN {X 0,Y 289.917,Z 453.225,A -85,B 0,C 180,E1 8464.946,E2 8464.946} C_VEL
LIN {X 0,Y 288.306,Z 449.741,A -85,B 0,C 180,E1 8460.397,E2 8460.397} C_VEL
LIN {X 0,Y 288.127,Z 449.731,A -85,B 0,C 180,E1 8455.621,E2 8455.621} C_VEL
LIN {X 0,Y 289.676,Z 453.945,A -85,B 0,C 180,E1 8450.463,E2 8450.463} C_VEL
LIN {X 0,Y 291.225,Z 457.563,A -85,B 0,C 180,E1 8447.81,E2 8447.81} C_VEL
LIN {X 0,Y 293.463,Z 462.57,A -85,B 0,C 180,E1 8444.992,E2 8444.992} C_VEL
LIN {X 0,Y 296.247,Z 469.2,A -85,B 0,C 180,E1 8442.179,E2 8442.179} C_VEL
LIN {X 0,Y 283.38,Z 599.046,A -85,B 0,C 180,E1 8439.712,E2 8439.712} C_VEL
LIN {X 0,Y 279.531,Z 620.585,A -85,B 0,C 180,E1 8439.138,E2 8439.138} C_VEL
LIN {X 0,Y 274.578,Z 640.372,A -85,B 0,C 180,E1 8438.402,E2 8438.402} C_VEL
LIN {X 0,Y 268.061,Z 660.672,A -85,B 0,C 180,E1 8437.39,E2 8437.39} C_VEL
LIN {X 0,Y 260.685,Z 679.43,A -85,B 0,C 180,E1 8436.169,E2 8436.169} C_VEL
LIN {X 0,Y 251.97,Z 697.792,A -85,B 0,C 180,E1 8434.623,E2 8434.623} C_VEL
LIN {X 0,Y 242.357,Z 715.212,A -85,B 0,C 180,E1 8432.745,E2 8432.745} C_VEL
LIN {X 0,Y 231.536,Z 732.298,A -85,B 0,C 180,E1 8430.38,E2 8430.38} C_VEL
LIN {X 0,Y 220.831,Z 747.283,A -85,B 0,C 180,E1 8427.705,E2 8427.705} C_VEL
LIN {X 0,Y 209.207,Z 761.76,A -85,B 0,C 180,E1 8424.332,E2 8424.332} C_VEL
LIN {X 0,Y 198.127,Z 774.21,A -85,B 0,C 180,E1 8420.515,E2 8420.515} C_VEL
LIN {X 0,Y 186.945,Z 785.825,A -85,B 0,C 180,E1 8415.78,E2 8415.78} C_VEL
LIN {X 0,Y 177.066,Z 795.464,A -85,B 0,C 180,E1 8410.494,E2 8410.494} C_VEL
LIN {X 0,Y 168.342,Z 803.689,A -85,B 0,C 180,E1 8404.349,E2 8404.349} C_VEL
LIN {X 0,Y 161.213,Z 810.315,A -85,B 0,C 180,E1 8397.319,E2 8397.319} C_VEL
LIN {X 0,Y 156.294,Z 815.133,A -85,B 0,C 180,E1 8389.819,E2 8389.819} C_VEL
LIN {X 0,Y 153.453,Z 818.401,A -85,B 0,C 180,E1 8381.653,E2 8381.653} C_VEL
LIN {X 0,Y 152.517,Z 819.884,A -85,B 0,C 180,E1 8374.512,E2 8374.512} C_VEL
LIN {X 0,Y 152.41,Z 820.041,A -85,B 0,C 180,E1 8368.12,E2 8368.12} C_VEL
LIN {X 0,Y 152.905,Z 819.229,A -85,B 0,C 180,E1 8361.35,E2 8361.35} C_VEL
LIN {X 0,Y 154.701,Z 816.909,A -85,B 0,C 180,E1 8353.865,E2 8353.865} C_VEL
LIN {X 0,Y 158.783,Z 812.681,A -85,B 0,C 180,E1 8345.839,E2 8345.839} C_VEL
LIN {X 0,Y 164.948,Z 806.876,A -85,B 0,C 180,E1 8338.581,E2 8338.581} C_VEL
LIN {X 0,Y 173.275,Z 799.18,A -85,B 0,C 180,E1 8331.873,E2 8331.873} C_VEL
LIN {X 0,Y 183.041,Z 789.836,A -85,B 0,C 180,E1 8326.075,E2 8326.075} C_VEL
LIN {X 0,Y 193.184,Z 779.592,A -85,B 0,C 180,E1 8321.37,E2 8321.37} C_VEL
LIN {X 0,Y 204.446,Z 767.388,A -85,B 0,C 180,E1 8317.142,E2 8317.142} C_VEL
LIN {X 0,Y 215.267,Z 754.617,A -85,B 0,C 180,E1 8313.759,E2 8313.759} C_VEL
LIN {X 0,Y 226.741,Z 739.473,A -85,B 0,C 180,E1 8310.698,E2 8310.698} C_VEL
LIN {X 0,Y 237.245,Z 723.856,A -85,B 0,C 180,E1 8308.262,E2 8308.262} C_VEL
LIN {X 0,Y 247.768,Z 706.032,A -85,B 0,C 180,E1 8306.096,E2 8306.096} C_VEL
LIN {X 0,Y 256.918,Z 688.107,A -85,B 0,C 180,E1 8304.406,E2 8304.406} C_VEL
LIN {X 0,Y 265.061,Z 669.257,A -85,B 0,C 180,E1 8303.017,E2 8303.017} C_VEL
LIN {X 0,Y 272.196,Z 648.995,A -85,B 0,C 180,E1 8301.883,E2 8301.883} C_VEL
LIN {X 0,Y 277.916,Z 628.39,A -85,B 0,C 180,E1 8301.019,E2 8301.019} C_VEL
LIN {X 0,Y 282.383,Z 606.505,A -85,B 0,C 180,E1 8300.363,E2 8300.363} C_VEL
LIN {X 0,Y 285.27,Z 584.13,A -85,B 0,C 180,E1 8299.881,E2 8299.881} C_VEL
LIN {X 0,Y 296.393,Z 469.228,A -85,B 0,C 180,E1 8297.675,E2 8297.675} C_VEL
LIN {X 0,Y 293.48,Z 462.345,A -85,B 0,C 180,E1 8294.704,E2 8294.704} C_VEL
LIN {X 0,Y 290.95,Z 456.408,A -85,B 0,C 180,E1 8291.297,E2 8291.297} C_VEL
LIN {X 0,Y 289.405,Z 453.055,A -85,B 0,C 180,E1 8288.344,E2 8288.344} C_VEL
LIN {X 0,Y 288.317,Z 449.821,A -85,B 0,C 180,E1 8283.778,E2 8283.778} C_VEL
LIN {X 0,Y 288.594,Z 449.992,A -85,B 0,C 180,E1 8279.405,E2 8279.405} C_VEL
LIN {X 0,Y 290.572,Z 454.262,A -85,B 0,C 180,E1 8274.273,E2 8274.273} C_VEL
LIN {X 0,Y 292.63,Z 458.552,A -85,B 0,C 180,E1 8271.255,E2 8271.255} C_VEL
LIN {X 0,Y 295.278,Z 463.994,A -85,B 0,C 180,E1 8268.328,E2 8268.328} C_VEL
LIN {X 0,Y 297.177,Z 468.376,A -85,B 0,C 180,E1 8266.539,E2 8266.539} C_VEL
LIN {X 0,Y 295.583,Z 483.996,A -85,B 0,C 180,E1 8266.24,E2 8266.24} C_VEL
LIN {X 0,Y 294.526,Z 491.686,A -85,B 0,C 180,E1 8266.277,E2 8266.277} C_VEL
LIN {X 0,Y 290.734,Z 512.203,A -85,B 0,C 180,E1 8267.063,E2 8267.063} C_VEL
LIN {X 0,Y 289.849,Z 518.805,A -85,B 0,C 180,E1 8267.085,E2 8267.085} C_VEL
LIN {X 0,Y 281.012,Z 601.988,A -85,B 0,C 180,E1 8265.463,E2 8265.463} C_VEL
LIN {X 0,Y 276.832,Z 624.269,A -85,B 0,C 180,E1 8264.895,E2 8264.895} C_VEL
LIN {X 0,Y 271.237,Z 645.455,A -85,B 0,C 180,E1 8264.174,E2 8264.174} C_VEL
LIN {X 0,Y 263.974,Z 666.956,A -85,B 0,C 180,E1 8263.166,E2 8263.166} C_VEL
LIN {X 0,Y 256.034,Z 686.252,A -85,B 0,C 180,E1 8261.968,E2 8261.968} C_VEL
LIN {X 0,Y 246.282,Z 706.135,A -85,B 0,C 180,E1 8260.365,E2 8260.365} C_VEL
LIN {X 0,Y 235.935,Z 724.168,A -85,B 0,C 180,E1 8258.463,E2 8258.463} C_VEL
LIN {X 0,Y 224.629,Z 741.501,A -85,B 0,C 180,E1 8256.106,E2 8256.106} C_VEL
LIN {X 0,Y 212.772,Z 757.721,A -85,B 0,C 180,E1 8253.23,E2 8253.23} C_VEL
LIN {X 0,Y 200.816,Z 772.512,A -85,B 0,C 180,E1 8249.81,E2 8249.81} C_VEL
LIN {X 0,Y 188.858,Z 785.955,A -85,B 0,C 180,E1 8245.678,E2 8245.678} C_VEL
LIN {X 0,Y 177.766,Z 797.646,A -85,B 0,C 180,E1 8240.911,E2 8240.911} C_VEL
LIN {X 0,Y 167.381,Z 808.193,A -85,B 0,C 180,E1 8235.181,E2 8235.181} C_VEL
LIN {X 0,Y 158.166,Z 817.516,A -85,B 0,C 180,E1 8228.279,E2 8228.279} C_VEL
LIN {X 0,Y 151.184,Z 824.889,A -85,B 0,C 180,E1 8220.612,E2 8220.612} C_VEL
LIN {X 0,Y 146.679,Z 830.436,A -85,B 0,C 180,E1 8212.44,E2 8212.44} C_VEL
LIN {X 0,Y 144.594,Z 834.143,A -85,B 0,C 180,E1 8204.414,E2 8204.414} C_VEL
LIN {X 0,Y 144.207,Z 836.063,A -85,B 0,C 180,E1 8197.169,E2 8197.169} C_VEL
LIN {X 0,Y 144.329,Z 836.727,A -85,B 0,C 180,E1 8191.191,E2 8191.191} C_VEL
LIN {X 0,Y 144.246,Z 836.483,A -85,B 0,C 180,E1 8185.229,E2 8185.229} C_VEL
LIN {X 0,Y 144.341,Z 834.879,A -85,B 0,C 180,E1 8178.006,E2 8178.006} C_VEL
LIN {X 0,Y 145.848,Z 831.714,A -85,B 0,C 180,E1 8169.916,E2 8169.916} C_VEL
LIN {X 0,Y 149.636,Z 826.61,A -85,B 0,C 180,E1 8161.679,E2 8161.679} C_VEL
LIN {X 0,Y 155.915,Z 819.699,A -85,B 0,C 180,E1 8153.845,E2 8153.845} C_VEL
LIN {X 0,Y 164.192,Z 811.302,A -85,B 0,C 180,E1 8146.948,E2 8146.948} C_VEL
LIN {X 0,Y 174.352,Z 801.109,A -85,B 0,C 180,E1 8140.803,E2 8140.803} C_VEL
LIN {X 0,Y 185.755,Z 789.174,A -85,B 0,C 180,E1 8135.543,E2 8135.543} C_VEL
LIN {X 0,Y 197.57,Z 776.027,A -85,B 0,C 180,E1 8131.213,E2 8131.213} C_VEL
LIN {X 0,Y 209.968,Z 761.094,A -85,B 0,C 180,E1 8127.51,E2 8127.51} C_VEL
LIN {X 0,Y 221.559,Z 745.721,A -85,B 0,C 180,E1 8124.59,E2 8124.59} C_VEL
LIN {X 0,Y 232.639,Z 729.215,A -85,B 0,C 180,E1 8122.187,E2 8122.187} C_VEL
LIN {X 0,Y 243.343,Z 711.112,A -85,B 0,C 180,E1 8120.141,E2 8120.141} C_VEL
LIN {X 0,Y 253.498,Z 691.266,A -85,B 0,C 180,E1 8118.421,E2 8118.421} C_VEL
LIN {X 0,Y 261.619,Z 672.667,A -85,B 0,C 180,E1 8117.171,E2 8117.171} C_VEL
LIN {X 0,Y 269.033,Z 652.044,A -85,B 0,C 180,E1 8116.12,E2 8116.12} C_VEL
LIN {X 0,Y 274.936,Z 631.316,A -85,B 0,C 180,E1 8115.339,E2 8115.339} C_VEL
LIN {X 0,Y 279.706,Z 608.601,A -85,B 0,C 180,E1 8114.709,E2 8114.709} C_VEL
LIN {X 0,Y 282.864,Z 584.532,A -85,B 0,C 180,E1 8114.189,E2 8114.189} C_VEL
LIN {X 0,Y 294.362,Z 473.292,A -85,B 0,C 180,E1 8112.057,E2 8112.057} C_VEL
LIN {X 0,Y 291.628,Z 467.208,A -85,B 0,C 180,E1 8109.074,E2 8109.074} C_VEL
LIN {X 0,Y 289.992,Z 463.74,A -85,B 0,C 180,E1 8106.831,E2 8106.831} C_VEL
LIN {X 0,Y 288.714,Z 460.947,A -85,B 0,C 180,E1 8104.568,E2 8104.568} C_VEL
LIN {X 0,Y 287.287,Z 457.647,A -85,B 0,C 180,E1 8100.199,E2 8100.199} C_VEL
LIN {X 0,Y 287.153,Z 457.69,A -85,B 0,C 180,E1 8095.606,E2 8095.606} C_VEL
LIN {X 0,Y 288.545,Z 461.773,A -85,B 0,C 180,E1 8090.727,E2 8090.727} C_VEL
LIN {X 0,Y 289.909,Z 465.119,A -85,B 0,C 180,E1 8088.259,E2 8088.259} C_VEL
LIN {X 0,Y 292.039,Z 470.132,A -85,B 0,C 180,E1 8085.425,E2 8085.425} C_VEL
LIN {X 0,Y 293.678,Z 474.55,A -85,B 0,C 180,E1 8083.588,E2 8083.588} C_VEL
LIN {X 0,Y 280.972,Z 599.212,A -85,B 0,C 180,E1 8081.262,E2 8081.262} C_VEL
LIN {X 0,Y 277.033,Z 620.789,A -85,B 0,C 180,E1 8080.705,E2 8080.705} C_VEL
LIN {X 0,Y 271.931,Z 640.729,A -85,B 0,C 180,E1 8079.985,E2 8079.985} C_VEL
LIN {X 0,Y 265.482,Z 660.449,A -85,B 0,C 180,E1 8079.035,E2 8079.035} C_VEL
LIN {X 0,Y 257.982,Z 679.172,A -85,B 0,C 180,E1 8077.86,E2 8077.86} C_VEL
LIN {X 0,Y 248.898,Z 697.935,A -85,B 0,C 180,E1 8076.331,E2 8076.331} C_VEL
LIN {X 0,Y 239.203,Z 715.106,A -85,B 0,C 180,E1 8074.535,E2 8074.535} C_VEL
LIN {X 0,Y 228.591,Z 731.532,A -85,B 0,C 180,E1 8072.339,E2 8072.339} C_VEL
LIN {X 0,Y 217.597,Z 746.565,A -85,B 0,C 180,E1 8069.75,E2 8069.75} C_VEL
LIN {X 0,Y 206.012,Z 760.595,A -85,B 0,C 180,E1 8066.591,E2 8066.591} C_VEL
LIN {X 0,Y 194.434,Z 773.282,A -85,B 0,C 180,E1 8062.849,E2 8062.849} C_VEL
LIN {X 0,Y 183.158,Z 784.626,A -85,B 0,C 180,E1 8058.405,E2 8058.405} C_VEL
LIN {X 0,Y 172.289,Z 794.795,A -85,B 0,C 180,E1 8053.01,E2 8053.01} C_VEL
LIN {X 0,Y 162.549,Z 803.382,A -85,B 0,C 180,E1 8046.63,E2 8046.63} C_VEL
LIN {X 0,Y 155.007,Z 809.907,A -85,B 0,C 180,E1 8039.78,E2 8039.78} C_VEL
LIN {X 0,Y 149.125,Z 815.199,A -85,B 0,C 180,E1 8031.639,E2 8031.639} C_VEL
LIN {X 0,Y 145.876,Z 818.538,A -85,B 0,C 180,E1 8023.476,E2 8023.476} C_VEL
LIN {X 0,Y 144.624,Z 820.148,A -85,B 0,C 180,E1 8015.952,E2 8015.952} C_VEL
LIN {X 0,Y 144.418,Z 820.531,A -85,B 0,C 180,E1 8008.81,E2 8008.81} C_VEL
LIN {X 0,Y 144.814,Z 819.864,A -85,B 0,C 180,E1 8002.063,E2 8002.063} C_VEL
LIN {X 0,Y 146.688,Z 817.659,A -85,B 0,C 180,E1 7993.772,E2 7993.772} C_VEL
LIN {X 0,Y 150.672,Z 813.858,A -85,B 0,C 180,E1 7985.706,E2 7985.706} C_VEL
LIN {X 0,Y 157.352,Z 807.999,A -85,B 0,C 180,E1 7977.741,E2 7977.741} C_VEL
LIN {X 0,Y 166.028,Z 800.428,A -85,B 0,C 180,E1 7970.779,E2 7970.779} C_VEL
LIN {X 0,Y 175.633,Z 791.792,A -85,B 0,C 180,E1 7965.098,E2 7965.098} C_VEL
LIN {X 0,Y 187.309,Z 780.678,A -85,B 0,C 180,E1 7959.767,E2 7959.767} C_VEL
LIN {X 0,Y 198.994,Z 768.62,A -85,B 0,C 180,E1 7955.516,E2 7955.516} C_VEL
LIN {X 0,Y 210.894,Z 755.112,A -85,B 0,C 180,E1 7951.938,E2 7951.938} C_VEL
LIN {X 0,Y 222.742,Z 739.982,A -85,B 0,C 180,E1 7948.919,E2 7948.919} C_VEL
LIN {X 0,Y 233.553,Z 724.397,A -85,B 0,C 180,E1 7946.528,E2 7946.528} C_VEL
LIN {X 0,Y 244.336,Z 706.651,A -85,B 0,C 180,E1 7944.413,E2 7944.413} C_VEL
LIN {X 0,Y 253.723,Z 688.765,A -85,B 0,C 180,E1 7942.764,E2 7942.764} C_VEL
LIN {X 0,Y 262.046,Z 669.963,A -85,B 0,C 180,E1 7941.413,E2 7941.413} C_VEL
LIN {X 0,Y 269.186,Z 650.281,A -85,B 0,C 180,E1 7940.333,E2 7940.333} C_VEL
LIN {X 0,Y 275.248,Z 629.158,A -85,B 0,C 180,E1 7939.464,E2 7939.464} C_VEL
LIN {X 0,Y 279.752,Z 607.926,A -85,B 0,C 180,E1 7938.838,E2 7938.838} C_VEL
LIN {X 0,Y 282.734,Z 586.137,A -85,B 0,C 180,E1 7938.373,E2 7938.373} C_VEL
LIN {X 0,Y 293.838,Z 474.411,A -85,B 0,C 180,E1 7936.263,E2 7936.263} C_VEL
LIN {X 0,Y 291.158,Z 467.614,A -85,B 0,C 180,E1 7933.1,E2 7933.1} C_VEL
LIN {X 0,Y 289.267,Z 463.2,A -85,B 0,C 180,E1 7930.154,E2 7930.154} C_VEL
LIN {X 0,Y 288.273,Z 460.791,A -85,B 0,C 180,E1 7927.975,E2 7927.975} C_VEL
LIN {X 0,Y 287.341,Z 457.766,A -85,B 0,C 180,E1 7923.791,E2 7923.791} C_VEL
LIN {X 0,Y 287.574,Z 457.879,A -85,B 0,C 180,E1 7919.602,E2 7919.602} C_VEL
LIN {X 0,Y 289.395,Z 462.08,A -85,B 0,C 180,E1 7914.548,E2 7914.548} C_VEL
LIN {X 0,Y 291.301,Z 466.249,A -85,B 0,C 180,E1 7911.612,E2 7911.612} C_VEL
LIN {X 0,Y 293.704,Z 471.459,A -85,B 0,C 180,E1 7908.811,E2 7908.811} C_VEL
LIN {X 0,Y 294.539,Z 473.653,A -85,B 0,C 180,E1 7907.937,E2 7907.937} C_VEL
LIN {X 0,Y 289.849,Z 518.805,A -85,B 0,C 180,E1 7907.085,E2 7907.085} C_VEL
LIN {X 0,Y 288.787,Z 526.496,A -85,B 0,C 180,E1 7907.133,E2 7907.133} C_VEL
LIN {X 0,Y 285.05,Z 547.007,A -85,B 0,C 180,E1 7907.952,E2 7907.952} C_VEL
LIN {X 0,Y 284.165,Z 553.607,A -85,B 0,C 180,E1 7907.975,E2 7907.975} C_VEL
LIN {X 0,Y 278.722,Z 602.534,A -85,B 0,C 180,E1 7907.029,E2 7907.029} C_VEL
LIN {X 0,Y 274.437,Z 624.806,A -85,B 0,C 180,E1 7906.478,E2 7906.478} C_VEL
LIN {X 0,Y 268.731,Z 645.839,A -85,B 0,C 180,E1 7905.785,E2 7905.785} C_VEL
LIN {X 0,Y 261.336,Z 667.195,A -85,B 0,C 180,E1 7904.817,E2 7904.817} C_VEL
LIN {X 0,Y 253.189,Z 686.49,A -85,B 0,C 180,E1 7903.657,E2 7903.657} C_VEL
LIN {X 0,Y 243.653,Z 705.499,A -85,B 0,C 180,E1 7902.178,E2 7902.178} C_VEL
LIN {X 0,Y 233.011,Z 723.644,A -85,B 0,C 180,E1 7900.336,E2 7900.336} C_VEL
LIN {X 0,Y 221.49,Z 740.864,A -85,B 0,C 180,E1 7898.071,E2 7898.071} C_VEL
LIN {X 0,Y 209.955,Z 756.259,A -85,B 0,C 180,E1 7895.445,E2 7895.445} C_VEL
LIN {X 0,Y 197.797,Z 770.806,A -85,B 0,C 180,E1 7892.202,E2 7892.202} C_VEL
LIN {X 0,Y 185.666,Z 784.017,A -85,B 0,C 180,E1 7888.304,E2 7888.304} C_VEL
LIN {X 0,Y 173.246,Z 796.571,A -85,B 0,C 180,E1 7883.34,E2 7883.34} C_VEL
LIN {X 0,Y 162.283,Z 807.119,A -85,B 0,C 180,E1 7877.674,E2 7877.674} C_VEL
LIN {X 0,Y 152.582,Z 816.205,A -85,B 0,C 180,E1 7870.94,E2 7870.94} C_VEL
LIN {X 0,Y 145.036,Z 823.454,A -85,B 0,C 180,E1 7863.469,E2 7863.469} C_VEL
LIN {X 0,Y 139.649,Z 829.303,A -85,B 0,C 180,E1 7854.987,E2 7854.987} C_VEL
LIN {X 0,Y 136.927,Z 833.238,A -85,B 0,C 180,E1 7846.545,E2 7846.545} C_VEL
LIN {X 0,Y 136.208,Z 835.456,A -85,B 0,C 180,E1 7838.442,E2 7838.442} C_VEL
LIN {X 0,Y 136.313,Z 836.202,A -85,B 0,C 180,E1 7832.522,E2 7832.522} C_VEL
LIN {X 0,Y 136.313,Z 836.198,A -85,B 0,C 180,E1 7827.478,E2 7827.478} C_VEL
LIN {X 0,Y 136.21,Z 835.365,A -85,B 0,C 180,E1 7821.133,E2 7821.133} C_VEL
LIN {X 0,Y 137.101,Z 832.858,A -85,B 0,C 180,E1 7812.603,E2 7812.603} C_VEL
LIN {X 0,Y 140.121,Z 828.738,A -85,B 0,C 180,E1 7804.038,E2 7804.038} C_VEL
LIN {X 0,Y 145.684,Z 822.755,A -85,B 0,C 180,E1 7795.753,E2 7795.753} C_VEL
LIN {X 0,Y 153.897,Z 814.85,A -85,B 0,C 180,E1 7787.997,E2 7787.997} C_VEL
LIN {X 0,Y 163.902,Z 805.468,A -85,B 0,C 180,E1 7781.382,E2 7781.382} C_VEL
LIN {X 0,Y 175.113,Z 794.675,A -85,B 0,C 180,E1 7775.829,E2 7775.829} C_VEL
LIN {X 0,Y 187.037,Z 782.432,A -85,B 0,C 180,E1 7771.207,E2 7771.207} C_VEL
LIN {X 0,Y 199.264,Z 768.898,A -85,B 0,C 180,E1 7767.363,E2 7767.363} C_VEL
LIN {X 0,Y 211.507,Z 754.077,A -85,B 0,C 180,E1 7764.169,E2 7764.169} C_VEL
LIN {X 0,Y 223.519,Z 737.797,A -85,B 0,C 180,E1 7761.501,E2 7761.501} C_VEL
LIN {X 0,Y 234.713,Z 720.586,A -85,B 0,C 180,E1 7759.345,E2 7759.345} C_VEL
LIN {X 0,Y 245.362,Z 701.862,A -85,B 0,C 180,E1 7757.536,E2 7757.536} C_VEL
LIN {X 0,Y 254.493,Z 683.226,A -85,B 0,C 180,E1 7756.143,E2 7756.143} C_VEL
LIN {X 0,Y 262.614,Z 663.399,A -85,B 0,C 180,E1 7755.004,E2 7755.004} C_VEL
LIN {X 0,Y 269.353,Z 643.11,A -85,B 0,C 180,E1 7754.128,E2 7754.128} C_VEL
LIN {X 0,Y 275.102,Z 620.771,A -85,B 0,C 180,E1 7753.429,E2 7753.429} C_VEL
LIN {X 0,Y 279.003,Z 598.905,A -85,B 0,C 180,E1 7752.907,E2 7752.907} C_VEL
LIN {X 0,Y 291.882,Z 478.529,A -85,B 0,C 180,E1 7750.61,E2 7750.61} C_VEL
LIN {X 0,Y 289.319,Z 472.552,A -85,B 0,C 180,E1 7747.346,E2 7747.346} C_VEL
LIN {X 0,Y 287.621,Z 468.82,A -85,B 0,C 180,E1 7744.386,E2 7744.386} C_VEL
LIN {X 0,Y 286.272,Z 465.554,A -85,B 0,C 180,E1 7740,E2 7740} C_VEL
LIN {X 0,Y 286.173,Z 465.701,A -85,B 0,C 180,E1 7735.591,E2 7735.591} C_VEL
LIN {X 0,Y 287.42,Z 469.601,A -85,B 0,C 180,E1 7730.993,E2 7730.993} C_VEL
LIN {X 0,Y 288.723,Z 472.983,A -85,B 0,C 180,E1 7728.525,E2 7728.525} C_VEL
LIN {X 0,Y 290.663,Z 477.836,A -85,B 0,C 180,E1 7725.812,E2 7725.812} C_VEL
LIN {X 0,Y 291.303,Z 479.677,A -85,B 0,C 180,E1 7725.024,E2 7725.024} C_VEL
LIN {X 0,Y 278.774,Z 599.373,A -85,B 0,C 180,E1 7722.838,E2 7722.838} C_VEL
LIN {X 0,Y 274.747,Z 620.989,A -85,B 0,C 180,E1 7722.298,E2 7722.298} C_VEL
LIN {X 0,Y 269.489,Z 641.109,A -85,B 0,C 180,E1 7721.597,E2 7721.597} C_VEL
LIN {X 0,Y 262.782,Z 661.117,A -85,B 0,C 180,E1 7720.663,E2 7720.663} C_VEL
LIN {X 0,Y 255.083,Z 679.877,A -85,B 0,C 180,E1 7719.519,E2 7719.519} C_VEL
LIN {X 0,Y 245.799,Z 698.565,A -85,B 0,C 180,E1 7718.038,E2 7718.038} C_VEL
LIN {X 0,Y 235.869,Z 715.677,A -85,B 0,C 180,E1 7716.292,E2 7716.292} C_VEL
LIN {X 0,Y 224.577,Z 732.606,A -85,B 0,C 180,E1 7714.068,E2 7714.068} C_VEL
LIN {X 0,Y 212.89,Z 748.016,A -85,B 0,C 180,E1 7711.431,E2 7711.431} C_VEL
LIN {X 0,Y 200.233,Z 762.742,A -85,B 0,C 180,E1 7708.089,E2 7708.089} C_VEL
LIN {X 0,Y 188.301,Z 775.126,A -85,B 0,C 180,E1 7704.33,E2 7704.33} C_VEL
LIN {X 0,Y 176.028,Z 786.763,A -85,B 0,C 180,E1 7699.563,E2 7699.563} C_VEL
LIN {X 0,Y 165.065,Z 796.385,A -85,B 0,C 180,E1 7694.153,E2 7694.153} C_VEL
LIN {X 0,Y 155.216,Z 804.606,A -85,B 0,C 180,E1 7687.73,E2 7687.73} C_VEL
LIN {X 0,Y 147,Z 811.23,A -85,B 0,C 180,E1 7680.22,E2 7680.22} C_VEL
LIN {X 0,Y 141.193,Z 816.042,A -85,B 0,C 180,E1 7672.043,E2 7672.043} C_VEL
LIN {X 0,Y 137.737,Z 819.305,A -85,B 0,C 180,E1 7663.005,E2 7663.005} C_VEL
LIN {X 0,Y 136.571,Z 820.782,A -85,B 0,C 180,E1 7655.04,E2 7655.04} C_VEL
LIN {X 0,Y 136.439,Z 820.937,A -85,B 0,C 180,E1 7647.9,E2 7647.9} C_VEL
LIN {X 0,Y 137.059,Z 820.128,A -85,B 0,C 180,E1 7640.341,E2 7640.341} C_VEL
LIN {X 0,Y 139.27,Z 817.813,A -85,B 0,C 180,E1 7632.019,E2 7632.019} C_VEL
LIN {X 0,Y 144.157,Z 813.59,A -85,B 0,C 180,E1 7623.204,E2 7623.204} C_VEL
LIN {X 0,Y 151.338,Z 807.79,A -85,B 0,C 180,E1 7615.377,E2 7615.377} C_VEL
LIN {X 0,Y 160.82,Z 800.098,A -85,B 0,C 180,E1 7608.3,E2 7608.3} C_VEL
LIN {X 0,Y 171.731,Z 790.757,A -85,B 0,C 180,E1 7602.319,E2 7602.319} C_VEL
LIN {X 0,Y 182.888,Z 780.528,A -85,B 0,C 180,E1 7597.561,E2 7597.561} C_VEL
LIN {X 0,Y 195.113,Z 768.348,A -85,B 0,C 180,E1 7593.356,E2 7593.356} C_VEL
LIN {X 0,Y 206.743,Z 755.604,A -85,B 0,C 180,E1 7590.042,E2 7590.042} C_VEL
LIN {X 0,Y 218.965,Z 740.488,A -85,B 0,C 180,E1 7587.076,E2 7587.076} C_VEL
LIN {X 0,Y 230.081,Z 724.937,A -85,B 0,C 180,E1 7584.739,E2 7584.739} C_VEL
LIN {X 0,Y 241.122,Z 707.266,A -85,B 0,C 180,E1 7582.684,E2 7582.684} C_VEL
LIN {X 0,Y 250.742,Z 689.423,A -85,B 0,C 180,E1 7581.081,E2 7581.081} C_VEL
LIN {X 0,Y 259.533,Z 669.997,A -85,B 0,C 180,E1 7579.73,E2 7579.73} C_VEL
LIN {X 0,Y 266.701,Z 650.613,A -85,B 0,C 180,E1 7578.705,E2 7578.705} C_VEL
LIN {X 0,Y 272.923,Z 629.38,A -85,B 0,C 180,E1 7577.861,E2 7577.861} C_VEL
LIN {X 0,Y 277.54,Z 608.037,A -85,B 0,C 180,E1 7577.255,E2 7577.255} C_VEL
LIN {X 0,Y 280.59,Z 586.237,A -85,B 0,C 180,E1 7576.803,E2 7576.803} C_VEL
LIN {X 0,Y 291.502,Z 479.648,A -85,B 0,C 180,E1 7574.857,E2 7574.857} C_VEL
LIN {X 0,Y 289.327,Z 474.121,A -85,B 0,C 180,E1 7571.967,E2 7571.967} C_VEL
LIN {X 0,Y 287.982,Z 470.663,A -85,B 0,C 180,E1 7569.594,E2 7569.594} C_VEL
LIN {X 0,Y 287.153,Z 468.526,A -85,B 0,C 180,E1 7567.604,E2 7567.604} C_VEL
LIN {X 0,Y 286.348,Z 465.684,A -85,B 0,C 180,E1 7563.604,E2 7563.604} C_VEL
LIN {X 0,Y 286.589,Z 465.901,A -85,B 0,C 180,E1 7559.601,E2 7559.601} C_VEL
LIN {X 0,Y 288.231,Z 469.898,A -85,B 0,C 180,E1 7554.826,E2 7554.826} C_VEL
LIN {X 0,Y 289.983,Z 473.943,A -85,B 0,C 180,E1 7551.973,E2 7551.973} C_VEL
LIN {X 0,Y 292.095,Z 478.82,A -85,B 0,C 180,E1 7549.364,E2 7549.364} C_VEL
LIN {X 0,Y 284.165,Z 553.607,A -85,B 0,C 180,E1 7547.975,E2 7547.975} C_VEL
LIN {X 0,Y 283.11,Z 561.295,A -85,B 0,C 180,E1 7548.027,E2 7548.027} C_VEL
LIN {X 0,Y 279.458,Z 581.8,A -85,B 0,C 180,E1 7548.879,E2 7548.879} C_VEL
LIN {X 0,Y 278.573,Z 588.4,A -85,B 0,C 180,E1 7548.913,E2 7548.913} C_VEL
LIN {X 0,Y 275.342,Z 610.549,A -85,B 0,C 180,E1 7548.45,E2 7548.45} C_VEL
LIN {X 0,Y 270.479,Z 632.231,A -85,B 0,C 180,E1 7547.885,E2 7547.885} C_VEL
LIN {X 0,Y 264.082,Z 653.451,A -85,B 0,C 180,E1 7547.138,E2 7547.138} C_VEL
LIN {X 0,Y 256.392,Z 673.78,A -85,B 0,C 180,E1 7546.168,E2 7546.168} C_VEL
LIN {X 0,Y 247.456,Z 693.115,A -85,B 0,C 180,E1 7544.943,E2 7544.943} C_VEL
LIN {X 0,Y 237.335,Z 711.699,A -85,B 0,C 180,E1 7543.415,E2 7543.415} C_VEL
LIN {X 0,Y 225.716,Z 730.151,A -85,B 0,C 180,E1 7541.43,E2 7541.43} C_VEL
LIN {X 0,Y 213.989,Z 746.497,A -85,B 0,C 180,E1 7539.143,E2 7539.143} C_VEL
LIN {X 0,Y 201.079,Z 762.393,A -85,B 0,C 180,E1 7536.193,E2 7536.193} C_VEL
LIN {X 0,Y 188.016,Z 776.773,A -85,B 0,C 180,E1 7532.632,E2 7532.632} C_VEL
LIN {X 0,Y 175.106,Z 789.752,A -85,B 0,C 180,E1 7528.295,E2 7528.295} C_VEL
LIN {X 0,Y 163.335,Z 800.797,A -85,B 0,C 180,E1 7523.311,E2 7523.311} C_VEL
LIN {X 0,Y 151.859,Z 810.97,A -85,B 0,C 180,E1 7516.955,E2 7516.955} C_VEL
LIN {X 0,Y 142.405,Z 819.198,A -85,B 0,C 180,E1 7509.711,E2 7509.711} C_VEL
LIN {X 0,Y 134.713,Z 826.27,A -85,B 0,C 180,E1 7500.805,E2 7500.805} C_VEL
LIN {X 0,Y 130.202,Z 831.206,A -85,B 0,C 180,E1 7491.629,E2 7491.629} C_VEL
LIN {X 0,Y 128.429,Z 834.115,A -85,B 0,C 180,E1 7483.048,E2 7483.048} C_VEL
LIN {X 0,Y 128.264,Z 835.616,A -85,B 0,C 180,E1 7474.919,E2 7474.919} C_VEL
LIN {X 0,Y 128.349,Z 835.826,A -85,B 0,C 180,E1 7468.661,E2 7468.661} C_VEL
LIN {X 0,Y 128.218,Z 835.162,A -85,B 0,C 180,E1 7462.033,E2 7462.033} C_VEL
LIN {X 0,Y 128.846,Z 833.204,A -85,B 0,C 180,E1 7453.778,E2 7453.778} C_VEL
LIN {X 0,Y 131.67,Z 829.38,A -85,B 0,C 180,E1 7444.64,E2 7444.64} C_VEL
LIN {X 0,Y 137.495,Z 823.576,A -85,B 0,C 180,E1 7435.445,E2 7435.445} C_VEL
LIN {X 0,Y 145.463,Z 816.504,A -85,B 0,C 180,E1 7427.655,E2 7427.655} C_VEL
LIN {X 0,Y 156.221,Z 807.037,A -85,B 0,C 180,E1 7420.393,E2 7420.393} C_VEL
LIN {X 0,Y 167.748,Z 796.573,A -85,B 0,C 180,E1 7414.662,E2 7414.662} C_VEL
LIN {X 0,Y 180.711,Z 784.11,A -85,B 0,C 180,E1 7409.699,E2 7409.699} C_VEL
LIN {X 0,Y 193.293,Z 770.996,A -85,B 0,C 180,E1 7405.837,E2 7405.837} C_VEL
LIN {X 0,Y 206.646,Z 755.554,A -85,B 0,C 180,E1 7402.463,E2 7402.463} C_VEL
LIN {X 0,Y 218.955,Z 739.52,A -85,B 0,C 180,E1 7399.835,E2 7399.835} C_VEL
LIN {X 0,Y 230.864,Z 721.991,A -85,B 0,C 180,E1 7397.647,E2 7397.647} C_VEL
LIN {X 0,Y 241.704,Z 703.688,A -85,B 0,C 180,E1 7395.896,E2 7395.896} C_VEL
LIN {X 0,Y 251.454,Z 684.505,A -85,B 0,C 180,E1 7394.488,E2 7394.488} C_VEL
LIN {X 0,Y 259.536,Z 665.353,A -85,B 0,C 180,E1 7393.412,E2 7393.412} C_VEL
LIN {X 0,Y 266.802,Z 644.367,A -85,B 0,C 180,E1 7392.522,E2 7392.522} C_VEL
LIN {X 0,Y 272.582,Z 622.879,A -85,B 0,C 180,E1 7391.863,E2 7391.863} C_VEL
LIN {X 0,Y 276.755,Z 600.982,A -85,B 0,C 180,E1 7391.348,E2 7391.348} C_VEL
LIN {X 0,Y 289.599,Z 484.139,A -85,B 0,C 180,E1 7389.194,E2 7389.194} C_VEL
LIN {X 0,Y 287.6,Z 479.343,A -85,B 0,C 180,E1 7386.287,E2 7386.287} C_VEL
LIN {X 0,Y 286.437,Z 476.543,A -85,B 0,C 180,E1 7384.003,E2 7384.003} C_VEL
LIN {X 0,Y 285.297,Z 473.499,A -85,B 0,C 180,E1 7380,E2 7380} C_VEL
LIN {X 0,Y 285.174,Z 473.587,A -85,B 0,C 180,E1 7375.777,E2 7375.777} C_VEL
LIN {X 0,Y 286.31,Z 477.44,A -85,B 0,C 180,E1 7371.252,E2 7371.252} C_VEL
LIN {X 0,Y 287.499,Z 480.718,A -85,B 0,C 180,E1 7368.871,E2 7368.871} C_VEL
LIN {X 0,Y 289.095,Z 484.929,A -85,B 0,C 180,E1 7366.482,E2 7366.482} C_VEL
LIN {X 0,Y 276.79,Z 599.534,A -85,B 0,C 180,E1 7364.437,E2 7364.437} C_VEL
LIN {X 0,Y 272.688,Z 621.133,A -85,B 0,C 180,E1 7363.919,E2 7363.919} C_VEL
LIN {X 0,Y 267.308,Z 641.341,A -85,B 0,C 180,E1 7363.243,E2 7363.243} C_VEL
LIN {X 0,Y 260.254,Z 661.899,A -85,B 0,C 180,E1 7362.317,E2 7362.317} C_VEL
LIN {X 0,Y 252.403,Z 680.557,A -85,B 0,C 180,E1 7361.216,E2 7361.216} C_VEL
LIN {X 0,Y 242.741,Z 699.535,A -85,B 0,C 180,E1 7359.757,E2 7359.757} C_VEL
LIN {X 0,Y 232.764,Z 716.246,A -85,B 0,C 180,E1 7358.098,E2 7358.098} C_VEL
LIN {X 0,Y 221.184,Z 733.136,A -85,B 0,C 180,E1 7355.939,E2 7355.939} C_VEL
LIN {X 0,Y 209.159,Z 748.517,A -85,B 0,C 180,E1 7353.368,E2 7353.368} C_VEL
LIN {X 0,Y 196.835,Z 762.409,A -85,B 0,C 180,E1 7350.296,E2 7350.296} C_VEL
LIN {X 0,Y 184.41,Z 774.92,A -85,B 0,C 180,E1 7346.611,E2 7346.611} C_VEL
LIN {X 0,Y 171.527,Z 786.673,A -85,B 0,C 180,E1 7341.898,E2 7341.898} C_VEL
LIN {X 0,Y 159.919,Z 796.405,A -85,B 0,C 180,E1 7336.489,E2 7336.489} C_VEL
LIN {X 0,Y 149.361,Z 804.695,A -85,B 0,C 180,E1 7329.988,E2 7329.988} C_VEL
LIN {X 0,Y 140.789,Z 811.11,A -85,B 0,C 180,E1 7322.665,E2 7322.665} C_VEL
LIN {X 0,Y 134.225,Z 816.107,A -85,B 0,C 180,E1 7314.185,E2 7314.185} C_VEL
LIN {X 0,Y 130.268,Z 819.442,A -85,B 0,C 180,E1 7305.127,E2 7305.127} C_VEL
LIN {X 0,Y 128.707,Z 821.047,A -85,B 0,C 180,E1 7296.692,E2 7296.692} C_VEL
LIN {X 0,Y 128.443,Z 821.427,A -85,B 0,C 180,E1 7288.662,E2 7288.662} C_VEL
LIN {X 0,Y 128.949,Z 820.763,A -85,B 0,C 180,E1 7281.079,E2 7281.079} C_VEL
LIN {X 0,Y 131.273,Z 818.564,A -85,B 0,C 180,E1 7271.804,E2 7271.804} C_VEL
LIN {X 0,Y 136.077,Z 814.767,A -85,B 0,C 180,E1 7262.9,E2 7262.9} C_VEL
LIN {X 0,Y 143.892,Z 808.91,A -85,B 0,C 180,E1 7254.291,E2 7254.291} C_VEL
LIN {X 0,Y 153.796,Z 801.341,A -85,B 0,C 180,E1 7246.952,E2 7246.952} C_VEL
LIN {X 0,Y 164.545,Z 792.714,A -85,B 0,C 180,E1 7241.109,E2 7241.109} C_VEL
LIN {X 0,Y 177.391,Z 781.615,A -85,B 0,C 180,E1 7235.745,E2 7235.745} C_VEL
LIN {X 0,Y 190.062,Z 769.581,A -85,B 0,C 180,E1 7231.547,E2 7231.547} C_VEL
LIN {X 0,Y 202.828,Z 756.093,A -85,B 0,C 180,E1 7228.07,E2 7228.07} C_VEL
LIN {X 0,Y 215.423,Z 740.995,A -85,B 0,C 180,E1 7225.171,E2 7225.171} C_VEL
LIN {X 0,Y 226.84,Z 725.476,A -85,B 0,C 180,E1 7222.898,E2 7222.898} C_VEL
LIN {X 0,Y 237.721,Z 708.588,A -85,B 0,C 180,E1 7220.979,E2 7220.979} C_VEL
LIN {X 0,Y 247.552,Z 690.942,A -85,B 0,C 180,E1 7219.425,E2 7219.425} C_VEL
LIN {X 0,Y 256.218,Z 672.367,A -85,B 0,C 180,E1 7218.158,E2 7218.158} C_VEL
LIN {X 0,Y 263.679,Z 653.129,A -85,B 0,C 180,E1 7217.148,E2 7217.148} C_VEL
LIN {X 0,Y 270.024,Z 632.683,A -85,B 0,C 180,E1 7216.335,E2 7216.335} C_VEL
LIN {X 0,Y 274.991,Z 611.369,A -85,B 0,C 180,E1 7215.72,E2 7215.72} C_VEL
LIN {X 0,Y 278.32,Z 589.255,A -85,B 0,C 180,E1 7215.264,E2 7215.264} C_VEL
LIN {X 0,Y 289.288,Z 485.032,A -85,B 0,C 180,E1 7213.39,E2 7213.39} C_VEL
LIN {X 0,Y 287.209,Z 479.292,A -85,B 0,C 180,E1 7210.025,E2 7210.025} C_VEL
LIN {X 0,Y 286.042,Z 476.261,A -85,B 0,C 180,E1 7207.23,E2 7207.23} C_VEL
LIN {X 0,Y 285.358,Z 473.602,A -85,B 0,C 180,E1 7203.415,E2 7203.415} C_VEL
LIN {X 0,Y 285.576,Z 473.778,A -85,B 0,C 180,E1 7199.8,E2 7199.8} C_VEL
LIN {X 0,Y 287.03,Z 477.576,A -85,B 0,C 180,E1 7195.205,E2 7195.205} C_VEL
LIN {X 0,Y 288.745,Z 481.799,A -85,B 0,C 180,E1 7192.239,E2 7192.239} C_VEL
LIN {X 0,Y 289.799,Z 484.414,A -85,B 0,C 180,E1 7190.806,E2 7190.806} C_VEL
LIN {X 0,Y 278.573,Z 588.4,A -85,B 0,C 180,E1 7188.913,E2 7188.913} C_VEL
LIN {X 0,Y 277.406,Z 596.076,A -85,B 0,C 180,E1 7188.974,E2 7188.974} C_VEL
LIN {X 0,Y 272.843,Z 615.295,A -85,B 0,C 180,E1 7189.801,E2 7189.801} C_VEL
LIN {X 0,Y 270.968,Z 622.844,A -85,B 0,C 180,E1 7189.794,E2 7189.794} C_VEL
LIN {X 0,Y 265.171,Z 644.056,A -85,B 0,C 180,E1 7189.179,E2 7189.179} C_VEL
LIN {X 0,Y 257.781,Z 665.075,A -85,B 0,C 180,E1 7188.336,E2 7188.336} C_VEL
LIN {X 0,Y 249.55,Z 684.226,A -85,B 0,C 180,E1 7187.315,E2 7187.315} C_VEL
LIN {X 0,Y 239.604,Z 703.405,A -85,B 0,C 180,E1 7185.974,E2 7185.974} C_VEL
LIN {X 0,Y 228.489,Z 721.755,A -85,B 0,C 180,E1 7184.299,E2 7184.299} C_VEL
LIN {X 0,Y 215.881,Z 739.788,A -85,B 0,C 180,E1 7182.129,E2 7182.129} C_VEL
LIN {X 0,Y 203.641,Z 755.237,A -85,B 0,C 180,E1 7179.679,E2 7179.679} C_VEL
LIN {X 0,Y 189.797,Z 770.707,A -85,B 0,C 180,E1 7176.399,E2 7176.399} C_VEL
LIN {X 0,Y 176.749,Z 783.763,A -85,B 0,C 180,E1 7172.637,E2 7172.637} C_VEL
LIN {X 0,Y 163.163,Z 796.208,A -85,B 0,C 180,E1 7167.74,E2 7167.74} C_VEL
LIN {X 0,Y 150.809,Z 806.775,A -85,B 0,C 180,E1 7161.934,E2 7161.934} C_VEL
LIN {X 0,Y 139.426,Z 816.107,A -85,B 0,C 180,E1 7154.649,E2 7154.649} C_VEL
LIN {X 0,Y 130.377,Z 823.487,A -85,B 0,C 180,E1 7146.192,E2 7146.192} C_VEL
LIN {X 0,Y 124.173,Z 829.048,A -85,B 0,C 180,E1 7136.802,E2 7136.802} C_VEL
LIN {X 0,Y 121.02,Z 832.771,A -85,B 0,C 180,E1 7127.303,E2 7127.303} C_VEL
LIN {X 0,Y 120.225,Z 834.705,A -85,B 0,C 180,E1 7118.609,E2 7118.609} C_VEL
LIN {X 0,Y 120.348,Z 835.356,A -85,B 0,C 180,E1 7111.904,E2 7111.904} C_VEL
LIN {X 0,Y 120.29,Z 835.218,A -85,B 0,C 180,E1 7105.71,E2 7105.71} C_VEL
LIN {X 0,Y 120.377,Z 834.012,A -85,B 0,C 180,E1 7097.529,E2 7097.529} C_VEL
LIN {X 0,Y 122.115,Z 831.237,A -85,B 0,C 180,E1 7088.38,E2 7088.38} C_VEL
LIN {X 0,Y 127.053,Z 826.301,A -85,B 0,C 180,E1 7078.18,E2 7078.18} C_VEL
LIN {X 0,Y 134.342,Z 820.154,A -85,B 0,C 180,E1 7069.647,E2 7069.647} C_VEL
LIN {X 0,Y 144.626,Z 811.773,A -85,B 0,C 180,E1 7061.701,E2 7061.701} C_VEL
LIN {X 0,Y 156.545,Z 801.826,A -85,B 0,C 180,E1 7055.163,E2 7055.163} C_VEL
LIN {X 0,Y 169.437,Z 790.453,A -85,B 0,C 180,E1 7049.839,E2 7049.839} C_VEL
LIN {X 0,Y 182.796,Z 777.7,A -85,B 0,C 180,E1 7045.512,E2 7045.512} C_VEL
LIN {X 0,Y 196.247,Z 763.542,A -85,B 0,C 180,E1 7041.991,E2 7041.991} C_VEL
LIN {X 0,Y 209.067,Z 748.345,A -85,B 0,C 180,E1 7039.176,E2 7039.176} C_VEL
LIN {X 0,Y 221.485,Z 731.806,A -85,B 0,C 180,E1 7036.861,E2 7036.861} C_VEL
LIN {X 0,Y 232.899,Z 714.504,A -85,B 0,C 180,E1 7035.001,E2 7035.001} C_VEL
LIN {X 0,Y 243.646,Z 695.633,A -85,B 0,C 180,E1 7033.454,E2 7033.454} C_VEL
LIN {X 0,Y 252.728,Z 676.667,A -85,B 0,C 180,E1 7032.267,E2 7032.267} C_VEL
LIN {X 0,Y 260.999,Z 655.894,A -85,B 0,C 180,E1 7031.281,E2 7031.281} C_VEL
LIN {X 0,Y 267.545,Z 635.387,A -85,B 0,C 180,E1 7030.562,E2 7030.562} C_VEL
LIN {X 0,Y 272.754,Z 613.766,A -85,B 0,C 180,E1 7030,E2 7030} C_VEL
LIN {X 0,Y 276.248,Z 591.4,A -85,B 0,C 180,E1 7029.539,E2 7029.539} C_VEL
LIN {X 0,Y 287.444,Z 489.792,A -85,B 0,C 180,E1 7027.696,E2 7027.696} C_VEL
LIN {X 0,Y 285.98,Z 486.125,A -85,B 0,C 180,E1 7025.215,E2 7025.215} C_VEL
LIN {X 0,Y 285.183,Z 484.116,A -85,B 0,C 180,E1 7023.417,E2 7023.417} C_VEL
LIN {X 0,Y 284.277,Z 481.407,A -85,B 0,C 180,E1 7019.798,E2 7019.798} C_VEL
LIN {X 0,Y 284.19,Z 481.626,A -85,B 0,C 180,E1 7015.763,E2 7015.763} C_VEL
LIN {X 0,Y 285.202,Z 485.254,A -85,B 0,C 180,E1 7011.532,E2 7011.532} C_VEL
LIN {X 0,Y 286.334,Z 488.593,A -85,B 0,C 180,E1 7009.131,E2 7009.131} C_VEL
LIN {X 0,Y 287.028,Z 490.646,A -85,B 0,C 180,E1 7007.951,E2 7007.951} C_VEL
LIN {X 0,Y 275.025,Z 599.694,A -85,B 0,C 180,E1 7006.059,E2 7006.059} C_VEL
LIN {X 0,Y 270.824,Z 621.399,A -85,B 0,C 180,E1 7005.56,E2 7005.56} C_VEL
LIN {X 0,Y 265.364,Z 641.529,A -85,B 0,C 180,E1 7004.916,E2 7004.916} C_VEL
LIN {X 0,Y 258.315,Z 661.759,A -85,B 0,C 180,E1 7004.048,E2 7004.048} C_VEL
LIN {X 0,Y 250.391,Z 680.32,A -85,B 0,C 180,E1 7003.007,E2 7003.007} C_VEL
LIN {X 0,Y 240.716,Z 699.02,A -85,B 0,C 180,E1 7001.639,E2 7001.639} C_VEL
LIN {X 0,Y 230.325,Z 716.156,A -85,B 0,C 180,E1 7000.021,E2 7000.021} C_VEL
LIN {X 0,Y 218.612,Z 732.912,A -85,B 0,C 180,E1 6997.973,E2 6997.973} C_VEL
LIN {X 0,Y 206.491,Z 748.102,A -85,B 0,C 180,E1 6995.546,E2 6995.546} C_VEL
LIN {X 0,Y 193.741,Z 762.075,A -85,B 0,C 180,E1 6992.577,E2 6992.577} C_VEL
LIN {X 0,Y 180.827,Z 774.715,A -85,B 0,C 180,E1 6988.985,E2 6988.985} C_VEL
LIN {X 0,Y 168.012,Z 786.027,A -85,B 0,C 180,E1 6984.615,E2 6984.615} C_VEL
LIN {X 0,Y 155.674,Z 795.97,A -85,B 0,C 180,E1 6979.276,E2 6979.276} C_VEL
LIN {X 0,Y 144.05,Z 804.542,A -85,B 0,C 180,E1 6972.628,E2 6972.628} C_VEL
LIN {X 0,Y 134.442,Z 811.278,A -85,B 0,C 180,E1 6964.935,E2 6964.935} C_VEL
LIN {X 0,Y 126.89,Z 816.562,A -85,B 0,C 180,E1 6955.682,E2 6955.682} C_VEL
LIN {X 0,Y 122.515,Z 819.893,A -85,B 0,C 180,E1 6946.109,E2 6946.109} C_VEL
LIN {X 0,Y 120.755,Z 821.497,A -85,B 0,C 180,E1 6937.134,E2 6937.134} C_VEL
LIN {X 0,Y 120.456,Z 821.876,A -85,B 0,C 180,E1 6928.573,E2 6928.573} C_VEL
LIN {X 0,Y 121.031,Z 821.212,A -85,B 0,C 180,E1 6920.49,E2 6920.49} C_VEL
LIN {X 0,Y 123.631,Z 819.016,A -85,B 0,C 180,E1 6910.636,E2 6910.636} C_VEL
LIN {X 0,Y 128.921,Z 815.222,A -85,B 0,C 180,E1 6901.26,E2 6901.26} C_VEL
LIN {X 0,Y 136.939,Z 809.656,A -85,B 0,C 180,E1 6892.699,E2 6892.699} C_VEL
LIN {X 0,Y 146.865,Z 802.579,A -85,B 0,C 180,E1 6885.476,E2 6885.476} C_VEL
LIN {X 0,Y 158.697,Z 793.675,A -85,B 0,C 180,E1 6879.201,E2 6879.201} C_VEL
LIN {X 0,Y 171.402,Z 783.303,A -85,B 0,C 180,E1 6874.057,E2 6874.057} C_VEL
LIN {X 0,Y 184.459,Z 771.546,A -85,B 0,C 180,E1 6869.859,E2 6869.859} C_VEL
LIN {X 0,Y 197.572,Z 758.238,A -85,B 0,C 180,E1 6866.398,E2 6866.398} C_VEL
LIN {X 0,Y 210.479,Z 743.495,A -85,B 0,C 180,E1 6863.537,E2 6863.537} C_VEL
LIN {X 0,Y 222.995,Z 727.214,A -85,B 0,C 180,E1 6861.156,E2 6861.156} C_VEL
LIN {X 0,Y 234.112,Z 710.624,A -85,B 0,C 180,E1 6859.295,E2 6859.295} C_VEL
LIN {X 0,Y 244.571,Z 692.365,A -85,B 0,C 180,E1 6857.725,E2 6857.725} C_VEL
LIN {X 0,Y 253.425,Z 674.015,A -85,B 0,C 180,E1 6856.504,E2 6856.504} C_VEL
LIN {X 0,Y 261.444,Z 653.975,A -85,B 0,C 180,E1 6855.482,E2 6855.482} C_VEL
LIN {X 0,Y 267.903,Z 633.759,A -85,B 0,C 180,E1 6854.706,E2 6854.706} C_VEL
LIN {X 0,Y 273.059,Z 612.2,A -85,B 0,C 180,E1 6854.105,E2 6854.105} C_VEL
LIN {X 0,Y 276.457,Z 590.458,A -85,B 0,C 180,E1 6853.669,E2 6853.669} C_VEL
LIN {X 0,Y 287.244,Z 490.628,A -85,B 0,C 180,E1 6851.906,E2 6851.906} C_VEL
LIN {X 0,Y 285.701,Z 486.182,A -85,B 0,C 180,E1 6848.96,E2 6848.96} C_VEL
LIN {X 0,Y 284.932,Z 483.996,A -85,B 0,C 180,E1 6846.853,E2 6846.853} C_VEL
LIN {X 0,Y 284.37,Z 481.521,A -85,B 0,C 180,E1 6843.225,E2 6843.225} C_VEL
LIN {X 0,Y 284.588,Z 481.816,A -85,B 0,C 180,E1 6839.799,E2 6839.799} C_VEL
LIN {X 0,Y 285.882,Z 485.391,A -85,B 0,C 180,E1 6835.487,E2 6835.487} C_VEL
LIN {X 0,Y 287.385,Z 489.327,A -85,B 0,C 180,E1 6832.705,E2 6832.705} C_VEL
LIN {X 0,Y 287.644,Z 490.307,A -85,B 0,C 180,E1 6832.265,E2 6832.265} C_VEL
LIN {X 0,Y 275.184,Z 601.217,A -85,B 0,C 180,E1 6830.282,E2 6830.282} C_VEL
LIN {X 0,Y 270.968,Z 622.844,A -85,B 0,C 180,E1 6829.794,E2 6829.794} C_VEL
LIN {X 0,Y 268.947,Z 630.344,A -85,B 0,C 180,E1 6829.806,E2 6829.806} C_VEL
LIN {X 0,Y 262.103,Z 648.984,A -85,B 0,C 180,E1 6830.516,E2 6830.516} C_VEL
LIN {X 0,Y 259.325,Z 656.219,A -85,B 0,C 180,E1 6830.445,E2 6830.445} C_VEL
LIN {X 0,Y 251.132,Z 676.405,A -85,B 0,C 180,E1 6829.54,E2 6829.54} C_VEL
LIN {X 0,Y 241.885,Z 695.363,A -85,B 0,C 180,E1 6828.418,E2 6828.418} C_VEL
LIN {X 0,Y 230.922,Z 714.229,A -85,B 0,C 180,E1 6826.954,E2 6826.954} C_VEL
LIN {X 0,Y 219.25,Z 731.523,A -85,B 0,C 180,E1 6825.188,E2 6825.188} C_VEL
LIN {X 0,Y 206.08,Z 748.563,A -85,B 0,C 180,E1 6822.897,E2 6822.897} C_VEL
LIN {X 0,Y 193.31,Z 763.223,A -85,B 0,C 180,E1 6820.277,E2 6820.277} C_VEL
LIN {X 0,Y 179.389,Z 777.368,A -85,B 0,C 180,E1 6816.873,E2 6816.873} C_VEL
LIN {X 0,Y 165.462,Z 790.101,A -85,B 0,C 180,E1 6812.657,E2 6812.657} C_VEL
LIN {X 0,Y 151.231,Z 801.993,A -85,B 0,C 180,E1 6807.101,E2 6807.101} C_VEL
LIN {X 0,Y 138.641,Z 811.811,A -85,B 0,C 180,E1 6800.502,E2 6800.502} C_VEL
LIN {X 0,Y 127.657,Z 820.115,A -85,B 0,C 180,E1 6792.343,E2 6792.343} C_VEL
LIN {X 0,Y 119.444,Z 826.43,A -85,B 0,C 180,E1 6782.963,E2 6782.963} C_VEL
LIN {X 0,Y 114.343,Z 830.986,A -85,B 0,C 180,E1 6772.628,E2 6772.628} C_VEL
LIN {X 0,Y 112.366,Z 833.781,A -85,B 0,C 180,E1 6762.331,E2 6762.331} C_VEL
LIN {X 0,Y 112.305,Z 834.8,A -85,B 0,C 180,E1 6754.084,E2 6754.084} C_VEL
LIN {X 0,Y 112.356,Z 834.903,A -85,B 0,C 180,E1 6747.96,E2 6747.96} C_VEL
LIN {X 0,Y 112.237,Z 834.238,A -85,B 0,C 180,E1 6740.773,E2 6740.773} C_VEL
LIN {X 0,Y 113.348,Z 832.158,A -85,B 0,C 180,E1 6730.951,E2 6730.951} C_VEL
LIN {X 0,Y 117.385,Z 828.095,A -85,B 0,C 180,E1 6720.395,E2 6720.395} C_VEL
LIN {X 0,Y 124.58,Z 822.315,A -85,B 0,C 180,E1 6710.652,E2 6710.652} C_VEL
LIN {X 0,Y 134.155,Z 815.131,A -85,B 0,C 180,E1 6702.453,E2 6702.453} C_VEL
LIN {X 0,Y 145.969,Z 806.087,A -85,B 0,C 180,E1 6695.403,E2 6695.403} C_VEL
LIN {X 0,Y 158.871,Z 795.608,A -85,B 0,C 180,E1 6689.717,E2 6689.717} C_VEL
LIN {X 0,Y 173.076,Z 783.123,A -85,B 0,C 180,E1 6684.912,E2 6684.912} C_VEL
LIN {X 0,Y 186.663,Z 769.977,A -85,B 0,C 180,E1 6681.251,E2 6681.251} C_VEL
LIN {X 0,Y 200.914,Z 754.522,A -85,B 0,C 180,E1 6678.104,E2 6678.104} C_VEL
LIN {X 0,Y 213.931,Z 738.432,A -85,B 0,C 180,E1 6675.685,E2 6675.685} C_VEL
LIN {X 0,Y 225.948,Z 721.55,A -85,B 0,C 180,E1 6673.761,E2 6673.761} C_VEL
LIN {X 0,Y 236.832,Z 704.046,A -85,B 0,C 180,E1 6672.226,E2 6672.226} C_VEL
LIN {X 0,Y 246.952,Z 684.969,A -85,B 0,C 180,E1 6670.947,E2 6670.947} C_VEL
LIN {X 0,Y 255.317,Z 666.045,A -85,B 0,C 180,E1 6669.976,E2 6669.976} C_VEL
LIN {X 0,Y 263.031,Z 644.713,A -85,B 0,C 180,E1 6669.155,E2 6669.155} C_VEL
LIN {X 0,Y 268.987,Z 623.48,A -85,B 0,C 180,E1 6668.565,E2 6668.565} C_VEL
LIN {X 0,Y 273.392,Z 601.353,A -85,B 0,C 180,E1 6668.087,E2 6668.087} C_VEL
LIN {X 0,Y 285.51,Z 495.68,A -85,B 0,C 180,E1 6666.245,E2 6666.245} C_VEL
LIN {X 0,Y 284.189,Z 492.14,A -85,B 0,C 180,E1 6663.429,E2 6663.429} C_VEL
LIN {X 0,Y 283.26,Z 489.319,A -85,B 0,C 180,E1 6659.595,E2 6659.595} C_VEL
LIN {X 0,Y 283.193,Z 489.517,A -85,B 0,C 180,E1 6655.95,E2 6655.95} C_VEL
LIN {X 0,Y 284.106,Z 493.077,A -85,B 0,C 180,E1 6651.805,E2 6651.805} C_VEL
LIN {X 0,Y 285.149,Z 496.387,A -85,B 0,C 180,E1 6649.442,E2 6649.442} C_VEL
LIN {X 0,Y 273.482,Z 599.852,A -85,B 0,C 180,E1 6647.7,E2 6647.7} C_VEL
LIN {X 0,Y 269.215,Z 621.524,A -85,B 0,C 180,E1 6647.225,E2 6647.225} C_VEL
LIN {X 0,Y 263.669,Z 641.652,A -85,B 0,C 180,E1 6646.614,E2 6646.614} C_VEL
LIN {X 0,Y 256.381,Z 662.195,A -85,B 0,C 180,E1 6645.777,E2 6645.777} C_VEL
LIN {X 0,Y 248.178,Z 681.002,A -85,B 0,C 180,E1 6644.768,E2 6644.768} C_VEL
LIN {X 0,Y 238.319,Z 699.648,A -85,B 0,C 180,E1 6643.463,E2 6643.463} C_VEL
LIN {X 0,Y 227.712,Z 716.726,A -85,B 0,C 180,E1 6641.915,E2 6641.915} C_VEL
LIN {X 0,Y 215.62,Z 733.578,A -85,B 0,C 180,E1 6639.931,E2 6639.931} C_VEL
LIN {X 0,Y 203.292,Z 748.607,A -85,B 0,C 180,E1 6637.611,E2 6637.611} C_VEL
LIN {X 0,Y 190.161,Z 762.567,A -85,B 0,C 180,E1 6634.735,E2 6634.735} C_VEL
LIN {X 0,Y 176.797,Z 775.192,A -85,B 0,C 180,E1 6631.23,E2 6631.23} C_VEL
LIN {X 0,Y 163.458,Z 786.495,A -85,B 0,C 180,E1 6626.929,E2 6626.929} C_VEL
LIN {X 0,Y 150.511,Z 796.433,A -85,B 0,C 180,E1 6621.616,E2 6621.616} C_VEL
LIN {X 0,Y 138.427,Z 804.836,A -85,B 0,C 180,E1 6615.059,E2 6615.059} C_VEL
LIN {X 0,Y 128.149,Z 811.559,A -85,B 0,C 180,E1 6607.264,E2 6607.264} C_VEL
LIN {X 0,Y 119.957,Z 816.822,A -85,B 0,C 180,E1 6597.824,E2 6597.824} C_VEL
LIN {X 0,Y 114.958,Z 820.241,A -85,B 0,C 180,E1 6587.723,E2 6587.723} C_VEL
LIN {X 0,Y 112.865,Z 821.884,A -85,B 0,C 180,E1 6578.148,E2 6578.148} C_VEL
LIN {X 0,Y 112.466,Z 822.345,A -85,B 0,C 180,E1 6568.981,E2 6568.981} C_VEL
LIN {X 0,Y 113.05,Z 821.724,A -85,B 0,C 180,E1 6560.326,E2 6560.326} C_VEL
LIN {X 0,Y 115.649,Z 819.767,A -85,B 0,C 180,E1 6550.296,E2 6550.296} C_VEL
LIN {X 0,Y 121.198,Z 816.123,A -85,B 0,C 180,E1 6540.332,E2 6540.332} C_VEL
LIN {X 0,Y 129.632,Z 810.689,A -85,B 0,C 180,E1 6531.337,E2 6531.337} C_VEL
LIN {X 0,Y 140.615,Z 803.426,A -85,B 0,C 180,E1 6523.509,E2 6523.509} C_VEL
LIN {X 0,Y 153.701,Z 794.135,A -85,B 0,C 180,E1 6516.859,E2 6516.859} C_VEL
LIN {X 0,Y 166.984,Z 783.788,A -85,B 0,C 180,E1 6511.763,E2 6511.763} C_VEL
LIN {X 0,Y 180.571,Z 772.018,A -85,B 0,C 180,E1 6507.634,E2 6507.634} C_VEL
LIN {X 0,Y 194.122,Z 758.724,A -85,B 0,C 180,E1 6504.267,E2 6504.267} C_VEL
LIN {X 0,Y 207.467,Z 743.921,A -85,B 0,C 180,E1 6501.486,E2 6501.486} C_VEL
LIN {X 0,Y 220.226,Z 727.753,A -85,B 0,C 180,E1 6499.209,E2 6499.209} C_VEL
LIN {X 0,Y 231.59,Z 711.211,A -85,B 0,C 180,E1 6497.425,E2 6497.425} C_VEL
LIN {X 0,Y 242.258,Z 692.981,A -85,B 0,C 180,E1 6495.925,E2 6495.925} C_VEL
LIN {X 0,Y 251.373,Z 674.507,A -85,B 0,C 180,E1 6494.748,E2 6494.748} C_VEL
LIN {X 0,Y 259.433,Z 654.819,A -85,B 0,C 180,E1 6493.788,E2 6493.788} C_VEL
LIN {X 0,Y 266.093,Z 634.483,A -85,B 0,C 180,E1 6493.041,E2 6493.041} C_VEL
LIN {X 0,Y 271.353,Z 612.946,A -85,B 0,C 180,E1 6492.467,E2 6492.467} C_VEL
LIN {X 0,Y 274.839,Z 591.444,A -85,B 0,C 180,E1 6492.05,E2 6492.05} C_VEL
LIN {X 0,Y 285.386,Z 496.557,A -85,B 0,C 180,E1 6490.446,E2 6490.446} C_VEL
LIN {X 0,Y 284.348,Z 493.273,A -85,B 0,C 180,E1 6488.086,E2 6488.086} C_VEL
LIN {X 0,Y 283.463,Z 490.193,A -85,B 0,C 180,E1 6484.451,E2 6484.451} C_VEL
LIN {X 0,Y 283.378,Z 489.422,A -85,B 0,C 180,E1 6482.832,E2 6482.832} C_VEL
LIN {X 0,Y 283.576,Z 489.693,A -85,B 0,C 180,E1 6480,E2 6480} C_VEL
LIN {X 0,Y 284.742,Z 493.206,A -85,B 0,C 180,E1 6475.772,E2 6475.772} C_VEL
LIN {X 0,Y 285.711,Z 496.06,A -85,B 0,C 180,E1 6473.748,E2 6473.748} C_VEL
LIN {X 0,Y 273.637,Z 601.287,A -85,B 0,C 180,E1 6471.924,E2 6471.924} C_VEL
LIN {X 0,Y 269.224,Z 623.441,A -85,B 0,C 180,E1 6471.446,E2 6471.446} C_VEL
LIN {X 0,Y 263.298,Z 644.585,A -85,B 0,C 180,E1 6470.861,E2 6470.861} C_VEL
LIN {X 0,Y 259.325,Z 656.219,A -85,B 0,C 180,E1 6470.445,E2 6470.445} C_VEL
LIN {X 0,Y 256.407,Z 663.467,A -85,B 0,C 180,E1 6470.366,E2 6470.366} C_VEL
LIN {X 0,Y 247.397,Z 681.313,A -85,B 0,C 180,E1 6470.863,E2 6470.863} C_VEL
LIN {X 0,Y 243.797,Z 688.094,A -85,B 0,C 180,E1 6470.719,E2 6470.719} C_VEL
LIN {X 0,Y 233.383,Z 706.909,A -85,B 0,C 180,E1 6469.482,E2 6469.482} C_VEL
LIN {X 0,Y 221.398,Z 725.359,A -85,B 0,C 180,E1 6467.88,E2 6467.88} C_VEL
LIN {X 0,Y 208.715,Z 742.112,A -85,B 0,C 180,E1 6465.944,E2 6465.944} C_VEL
LIN {X 0,Y 195.008,Z 758.011,A -85,B 0,C 180,E1 6463.491,E2 6463.491} C_VEL
LIN {X 0,Y 180.458,Z 772.913,A -85,B 0,C 180,E1 6460.371,E2 6460.371} C_VEL
LIN {X 0,Y 166.205,Z 785.963,A -85,B 0,C 180,E1 6456.607,E2 6456.607} C_VEL
LIN {X 0,Y 151.203,Z 798.222,A -85,B 0,C 180,E1 6451.578,E2 6451.578} C_VEL
LIN {X 0,Y 137.973,Z 808.11,A -85,B 0,C 180,E1 6445.701,E2 6445.701} C_VEL
LIN {X 0,Y 125.308,Z 817.046,A -85,B 0,C 180,E1 6437.906,E2 6437.906} C_VEL
LIN {X 0,Y 115.286,Z 824.036,A -85,B 0,C 180,E1 6428.69,E2 6428.69} C_VEL
LIN {X 0,Y 108.345,Z 829.239,A -85,B 0,C 180,E1 6418.076,E2 6418.076} C_VEL
LIN {X 0,Y 104.936,Z 832.49,A -85,B 0,C 180,E1 6407.18,E2 6407.18} C_VEL
LIN {X 0,Y 104.25,Z 834.184,A -85,B 0,C 180,E1 6397.162,E2 6397.162} C_VEL
LIN {X 0,Y 104.406,Z 834.548,A -85,B 0,C 180,E1 6390,E2 6390} C_VEL
LIN {X 0,Y 104.242,Z 834.094,A -85,B 0,C 180,E1 6382.283,E2 6382.283} C_VEL
LIN {X 0,Y 105.035,Z 832.337,A -85,B 0,C 180,E1 6372.265,E2 6372.265} C_VEL
LIN {X 0,Y 108.961,Z 828.658,A -85,B 0,C 180,E1 6360.66,E2 6360.66} C_VEL
LIN {X 0,Y 116.08,Z 823.452,A -85,B 0,C 180,E1 6350.403,E2 6350.403} C_VEL
LIN {X 0,Y 126.406,Z 816.225,A -85,B 0,C 180,E1 6341.287,E2 6341.287} C_VEL
LIN {X 0,Y 138.625,Z 807.529,A -85,B 0,C 180,E1 6333.959,E2 6333.959} C_VEL
LIN {X 0,Y 152.673,Z 796.91,A -85,B 0,C 180,E1 6327.86,E2 6327.86} C_VEL
LIN {X 0,Y 166.54,Z 785.521,A -85,B 0,C 180,E1 6323.286,E2 6323.286} C_VEL
LIN {X 0,Y 181.29,Z 771.946,A -85,B 0,C 180,E1 6319.425,E2 6319.425} C_VEL
LIN {X 0,Y 194.999,Z 757.797,A -85,B 0,C 180,E1 6316.501,E2 6316.501} C_VEL
LIN {X 0,Y 209.155,Z 741.287,A -85,B 0,C 180,E1 6313.974,E2 6313.974} C_VEL
LIN {X 0,Y 221.847,Z 724.364,A -85,B 0,C 180,E1 6312.045,E2 6312.045} C_VEL
LIN {X 0,Y 233.375,Z 706.562,A -85,B 0,C 180,E1 6310.508,E2 6310.508} C_VEL
LIN {X 0,Y 243.652,Z 687.934,A -85,B 0,C 180,E1 6309.286,E2 6309.286} C_VEL
LIN {X 0,Y 252.914,Z 667.952,A -85,B 0,C 180,E1 6308.283,E2 6308.283} C_VEL
LIN {X 0,Y 260.456,Z 648.134,A -85,B 0,C 180,E1 6307.536,E2 6307.536} C_VEL
LIN {X 0,Y 266.882,Z 626.452,A -85,B 0,C 180,E1 6306.945,E2 6306.945} C_VEL
LIN {X 0,Y 271.446,Z 604.833,A -85,B 0,C 180,E1 6306.494,E2 6306.494} C_VEL
LIN {X 0,Y 275.455,Z 574.154,A -85,B 0,C 180,E1 6305.955,E2 6305.955} C_VEL
LIN {X 0,Y 283.713,Z 501.867,A -85,B 0,C 180,E1 6304.75,E2 6304.75} C_VEL
LIN {X 0,Y 282.964,Z 499.711,A -85,B 0,C 180,E1 6302.835,E2 6302.835} C_VEL
LIN {X 0,Y 282.245,Z 497.235,A -85,B 0,C 180,E1 6299.391,E2 6299.391} C_VEL
LIN {X 0,Y 282.194,Z 497.407,A -85,B 0,C 180,E1 6296.14,E2 6296.14} C_VEL
LIN {X 0,Y 283.009,Z 500.9,A -85,B 0,C 180,E1 6292.08,E2 6292.08} C_VEL
LIN {X 0,Y 283.422,Z 502.442,A -85,B 0,C 180,E1 6290.945,E2 6290.945} C_VEL
LIN {X 0,Y 272.167,Z 600.009,A -85,B 0,C 180,E1 6289.358,E2 6289.358} C_VEL
LIN {X 0,Y 267.816,Z 621.743,A -85,B 0,C 180,E1 6288.907,E2 6288.907} C_VEL
LIN {X 0,Y 262.32,Z 641.426,A -85,B 0,C 180,E1 6288.345,E2 6288.345} C_VEL
LIN {X 0,Y 255.408,Z 660.878,A -85,B 0,C 180,E1 6287.608,E2 6287.608} C_VEL
LIN {X 0,Y 247.073,Z 679.879,A -85,B 0,C 180,E1 6286.663,E2 6286.663} C_VEL
LIN {X 0,Y 237.529,Z 697.872,A -85,B 0,C 180,E1 6285.497,E2 6285.497} C_VEL
LIN {X 0,Y 226.18,Z 716.081,A -85,B 0,C 180,E1 6283.969,E2 6283.969} C_VEL
LIN {X 0,Y 214.266,Z 732.535,A -85,B 0,C 180,E1 6282.162,E2 6282.162} C_VEL
LIN {X 0,Y 201.224,Z 748.149,A -85,B 0,C 180,E1 6279.9,E2 6279.9} C_VEL
LIN {X 0,Y 187.238,Z 762.684,A -85,B 0,C 180,E1 6277.056,E2 6277.056} C_VEL
LIN {X 0,Y 173.052,Z 775.668,A -85,B 0,C 180,E1 6273.577,E2 6273.577} C_VEL
LIN {X 0,Y 158.44,Z 787.518,A -85,B 0,C 180,E1 6269.118,E2 6269.118} C_VEL
LIN {X 0,Y 144.935,Z 797.342,A -85,B 0,C 180,E1 6263.816,E2 6263.816} C_VEL
LIN {X 0,Y 131.945,Z 805.879,A -85,B 0,C 180,E1 6256.998,E2 6256.998} C_VEL
LIN {X 0,Y 121.027,Z 812.482,A -85,B 0,C 180,E1 6248.892,E2 6248.892} C_VEL
LIN {X 0,Y 112.525,Z 817.471,A -85,B 0,C 180,E1 6239.255,E2 6239.255} C_VEL
LIN {X 0,Y 107.122,Z 820.797,A -85,B 0,C 180,E1 6228.502,E2 6228.502} C_VEL
LIN {X 0,Y 104.874,Z 822.397,A -85,B 0,C 180,E1 6218.222,E2 6218.222} C_VEL
LIN {X 0,Y 104.479,Z 822.793,A -85,B 0,C 180,E1 6208.903,E2 6208.903} C_VEL
LIN {X 0,Y 105.15,Z 822.174,A -85,B 0,C 180,E1 6199.592,E2 6199.592} C_VEL
LIN {X 0,Y 108.085,Z 820.22,A -85,B 0,C 180,E1 6188.853,E2 6188.853} C_VEL
LIN {X 0,Y 114.231,Z 816.575,A -85,B 0,C 180,E1 6178.321,E2 6178.321} C_VEL
LIN {X 0,Y 123.402,Z 811.143,A -85,B 0,C 180,E1 6168.983,E2 6168.983} C_VEL
LIN {X 0,Y 135.156,Z 803.882,A -85,B 0,C 180,E1 6161.014,E2 6161.014} C_VEL
LIN {X 0,Y 148.283,Z 795.096,A -85,B 0,C 180,E1 6154.653,E2 6154.653} C_VEL
LIN {X 0,Y 162.264,Z 784.751,A -85,B 0,C 180,E1 6149.536,E2 6149.536} C_VEL
LIN {X 0,Y 176.969,Z 772.489,A -85,B 0,C 180,E1 6145.317,E2 6145.317} C_VEL
LIN {X 0,Y 190.951,Z 759.208,A -85,B 0,C 180,E1 6142.061,E2 6142.061} C_VEL
LIN {X 0,Y 204.587,Z 744.508,A -85,B 0,C 180,E1 6139.403,E2 6139.403} C_VEL
LIN {X 0,Y 217.276,Z 728.891,A -85,B 0,C 180,E1 6137.284,E2 6137.284} C_VEL
LIN {X 0,Y 229.32,Z 711.792,A -85,B 0,C 180,E1 6135.517,E2 6135.517} C_VEL
LIN {X 0,Y 240.188,Z 693.597,A -85,B 0,C 180,E1 6134.092,E2 6134.092} C_VEL
LIN {X 0,Y 249.558,Z 675.004,A -85,B 0,C 180,E1 6132.966,E2 6132.966} C_VEL
LIN {X 0,Y 257.653,Z 655.662,A -85,B 0,C 180,E1 6132.07,E2 6132.07} C_VEL
LIN {X 0,Y 264.546,Z 635.072,A -85,B 0,C 180,E1 6131.35,E2 6131.35} C_VEL
LIN {X 0,Y 269.897,Z 613.58,A -85,B 0,C 180,E1 6130.806,E2 6130.806} C_VEL
LIN {X 0,Y 273.486,Z 592.112,A -85,B 0,C 180,E1 6130.408,E2 6130.408} C_VEL
LIN {X 0,Y 283.674,Z 502.415,A -85,B 0,C 180,E1 6128.922,E2 6128.922} C_VEL
LIN {X 0,Y 282.801,Z 499.617,A -85,B 0,C 180,E1 6126.293,E2 6126.293} C_VEL
LIN {X 0,Y 282.412,Z 497.385,A -85,B 0,C 180,E1 6123.045,E2 6123.045} C_VEL
LIN {X 0,Y 282.561,Z 497.568,A -85,B 0,C 180,E1 6120.203,E2 6120.203} C_VEL
LIN {X 0,Y 283.609,Z 501.019,A -85,B 0,C 180,E1 6116.058,E2 6116.058} C_VEL
LIN {X 0,Y 283.918,Z 502.293,A -85,B 0,C 180,E1 6115.242,E2 6115.242} C_VEL
LIN {X 0,Y 272.346,Z 601.161,A -85,B 0,C 180,E1 6113.586,E2 6113.586} C_VEL
LIN {X 0,Y 267.876,Z 623.302,A -85,B 0,C 180,E1 6113.134,E2 6113.134} C_VEL
LIN {X 0,Y 261.894,Z 644.37,A -85,B 0,C 180,E1 6112.588,E2 6112.588} C_VEL
LIN {X 0,Y 254.042,Z 665.799,A -85,B 0,C 180,E1 6111.82,E2 6111.82} C_VEL
LIN {X 0,Y 245.542,Z 684.716,A -85,B 0,C 180,E1 6110.911,E2 6110.911} C_VEL
LIN {X 0,Y 243.797,Z 688.094,A -85,B 0,C 180,E1 6110.719,E2 6110.719} C_VEL
LIN {X 0,Y 240.048,Z 694.929,A -85,B 0,C 180,E1 6110.551,E2 6110.551} C_VEL
